LIN {X -0.007,Y -160.947,Z 1391.312,A 0.000,B 0.000,C 90.000,E1 236.135} C_DIS
LIN {X -0.022,Y -157.703,Z 1391.292,A 0.000,B 0.000,C 90.000,E1 232.603} C_DIS
LIN {X 0.041,Y -155.743,Z 1391.277,A 0.000,B 0.000,C 90.000,E1 229.908} C_DIS
LIN {X -0.013,Y -152.001,Z 1391.252,A 0.000,B 0.000,C 90.000,E1 225.445} C_DIS
LIN {X -0.001,Y -150.246,Z 1391.237,A 0.000,B 0.000,C 90.000,E1 222.732} C_DIS
LIN {X 0.031,Y -147.004,Z 1391.212,A 0.000,B 0.000,C 90.000,E1 218.177} C_DIS
LIN {X 0.021,Y -145.588,Z 1391.197,A 0.000,B 0.000,C 90.000,E1 215.438} C_DIS
LIN {X -0.058,Y -142.976,Z 1391.171,A 0.000,B 0.000,C 90.000,E1 210.875} C_DIS
LIN {X 0.069,Y -141.603,Z 1391.151,A 0.000,B 0.000,C 90.000,E1 207.129} C_DIS
LIN {X -0.017,Y -139.424,Z 1391.115,A 0.000,B 0.000,C 90.000,E1 200.663} C_DIS
LIN {X 0.035,Y -139.153,Z 1391.104,A 0.000,B 0.000,C 90.000,E1 198.779} C_DIS
LIN {X 0.057,Y -138.344,Z 1391.058,A 0.000,B 0.000,C 90.000,E1 190.366} C_DIS
LIN {X 0.043,Y -139.484,Z 1391.006,A 0.000,B 0.000,C 90.000,E1 181.031} C_DIS
LIN {X -0.017,Y -141.082,Z 1390.975,A 0.000,B 0.000,C 90.000,E1 175.469} C_DIS
LIN {X -0.063,Y -142.458,Z 1390.959,A 0.000,B 0.000,C 90.000,E1 172.704} C_DIS
LIN {X 0.027,Y -144.702,Z 1390.934,A 0.000,B 0.000,C 90.000,E1 168.049} C_DIS
LIN {X -0.021,Y -147.298,Z 1390.913,A 0.000,B 0.000,C 90.000,E1 164.393} C_DIS
LIN {X -0.007,Y -150.618,Z 1390.888,A 0.000,B 0.000,C 90.000,E1 159.826} C_DIS
LIN {X -0.071,Y -154.093,Z 1390.868,A 0.000,B 0.000,C 90.000,E1 156.230} C_DIS
LIN {X -0.006,Y -157.515,Z 1390.848,A 0.000,B 0.000,C 90.000,E1 152.615} C_DIS
LIN {X -0.061,Y -161.747,Z 1390.828,A 0.000,B 0.000,C 90.000,E1 149.076} C_DIS
LIN {X 0.045,Y -165.940,Z 1390.808,A 0.000,B 0.000,C 90.000,E1 145.515} C_DIS
LIN {X 0.043,Y -170.931,Z 1390.789,A 0.000,B 0.000,C 90.000,E1 142.029} C_DIS
LIN {X -0.037,Y -175.799,Z 1390.770,A 0.000,B 0.000,C 90.000,E1 138.609} C_DIS
LIN {X 0.091,Y -181.407,Z 1390.751,A 0.000,B 0.000,C 90.000,E1 135.162} C_DIS
LIN {X -0.034,Y -186.908,Z 1390.732,A 0.000,B 0.000,C 90.000,E1 131.838} C_DIS
LIN {X -0.082,Y -191.488,Z 1390.719,A 0.000,B 0.000,C 90.000,E1 129.358} C_DIS
LIN {X 0.125,Y -197.349,Z 1390.700,A 0.000,B 0.000,C 90.000,E1 126.011} C_DIS
LIN {X -0.018,Y -199.398,Z 1390.695,A 0.000,B 0.000,C 90.000,E1 125.025} C_DIS
LIN {X -0.063,Y -309.902,Z 1390.694,A 0.000,B 0.000,C 90.000,E1 125.025} C_DIS
LIN {X -0.002,Y -311.910,Z 1390.694,A 0.000,B 0.000,C 90.000,E1 124.978} C_DIS
LIN {X 0.038,Y -317.203,Z 1390.693,A 0.000,B 0.000,C 90.000,E1 124.692} C_DIS
LIN {X 0.080,Y -320.044,Z 1390.691,A 0.000,B 0.000,C 90.000,E1 124.405} C_DIS
LIN {X 0.017,Y -323.693,Z 1390.688,A 0.000,B 0.000,C 90.000,E1 123.865} C_DIS
LIN {X -0.171,Y -325.159,Z 1390.686,A 0.000,B 0.000,C 90.000,E1 123.579} C_DIS
LIN {X 0.060,Y -338.025,Z 1390.667,A 0.000,B 0.000,C 90.000,E1 120.079} C_DIS
LIN {X -0.098,Y -349.982,Z 1390.652,A 0.000,B 0.000,C 90.000,E1 117.334} C_DIS
LIN {X 0.073,Y -363.402,Z 1390.637,A 0.000,B 0.000,C 90.000,E1 114.591} C_DIS
LIN {X 0.224,Y -376.645,Z 1390.624,A 0.000,B 0.000,C 90.000,E1 112.206} C_DIS
LIN {X -0.078,Y -391.224,Z 1390.611,A 0.000,B 0.000,C 90.000,E1 109.939} C_DIS
LIN {X -0.169,Y -407.239,Z 1390.598,A 0.000,B 0.000,C 90.000,E1 107.692} C_DIS
LIN {X -0.119,Y -424.803,Z 1390.586,A 0.000,B 0.000,C 90.000,E1 105.481} C_DIS
LIN {X 0.188,Y -444.001,Z 1390.574,A 0.000,B 0.000,C 90.000,E1 103.300} C_DIS
LIN {X 0.222,Y -464.106,Z 1390.563,A 0.000,B 0.000,C 90.000,E1 101.299} C_DIS
LIN {X -0.112,Y -482.128,Z 1390.554,A 0.000,B 0.000,C 90.000,E1 99.726} C_DIS
LIN {X -0.082,Y -484.477,Z 1390.553,A 0.000,B 0.000,C 90.000,E1 99.500} C_DIS
LIN {X -0.092,Y -486.349,Z 1390.551,A 0.000,B 0.000,C 90.000,E1 99.265} C_DIS
LIN {X -0.103,Y -487.770,Z 1390.550,A 0.000,B 0.000,C 90.000,E1 99.029} C_DIS
LIN {X 0.094,Y -489.689,Z 1390.547,A 0.000,B 0.000,C 90.000,E1 98.511} C_DIS
LIN {X -0.183,Y -490.477,Z 1390.545,A 0.000,B 0.000,C 90.000,E1 98.049} C_DIS
LIN {X 0.039,Y -490.272,Z 1390.542,A 0.000,B 0.000,C 90.000,E1 97.530} C_DIS
LIN {X -0.220,Y -489.046,Z 1390.539,A 0.000,B 0.000,C 90.000,E1 97.068} C_DIS
LIN {X 0.164,Y -487.991,Z 1390.538,A 0.000,B 0.000,C 90.000,E1 96.777} C_DIS
LIN {X 0.006,Y -486.568,Z 1390.536,A 0.000,B 0.000,C 90.000,E1 96.549} C_DIS
LIN {X 0.174,Y -468.415,Z 1390.521,A 0.000,B 0.000,C 90.000,E1 93.784} C_DIS
LIN {X 0.105,Y -460.162,Z 1390.514,A 0.000,B 0.000,C 90.000,E1 92.522} C_DIS
LIN {X 0.170,Y -439.101,Z 1390.495,A 0.000,B 0.000,C 90.000,E1 89.141} C_DIS
LIN {X 0.130,Y -427.055,Z 1390.484,A 0.000,B 0.000,C 90.000,E1 87.020} C_DIS
LIN {X 0.051,Y -417.995,Z 1390.475,A 0.000,B 0.000,C 90.000,E1 85.412} C_DIS
LIN {X -0.076,Y -407.198,Z 1390.464,A 0.000,B 0.000,C 90.000,E1 83.514} C_DIS
LIN {X -0.007,Y -397.916,Z 1390.455,A 0.000,B 0.000,C 90.000,E1 81.837} C_DIS
LIN {X -0.041,Y -388.423,Z 1390.445,A 0.000,B 0.000,C 90.000,E1 80.151} C_DIS
LIN {X 0.150,Y -377.105,Z 1390.434,A 0.000,B 0.000,C 90.000,E1 78.117} C_DIS
LIN {X -0.100,Y -367.376,Z 1390.424,A 0.000,B 0.000,C 90.000,E1 76.408} C_DIS
LIN {X -0.068,Y -357.511,Z 1390.415,A 0.000,B 0.000,C 90.000,E1 74.629} C_DIS
LIN {X 0.139,Y -345.870,Z 1390.403,A 0.000,B 0.000,C 90.000,E1 72.489} C_DIS
LIN {X -0.034,Y -334.159,Z 1390.391,A 0.000,B 0.000,C 90.000,E1 70.369} C_DIS
LIN {X 0.000,Y -319.385,Z 1390.375,A 0.000,B 0.000,C 90.000,E1 67.539} C_DIS
LIN {X -0.087,Y -304.192,Z 1390.357,A 0.000,B 0.000,C 90.000,E1 64.332} C_DIS
LIN {X -0.089,Y -294.606,Z 1390.344,A 0.000,B 0.000,C 90.000,E1 62.025} C_DIS
LIN {X -0.064,Y -283.523,Z 1390.328,A 0.000,B 0.000,C 90.000,E1 58.997} C_DIS
LIN {X 0.029,Y -272.556,Z 1390.309,A 0.000,B 0.000,C 90.000,E1 55.548} C_DIS
LIN {X 0.000,Y -264.344,Z 1390.293,A 0.000,B 0.000,C 90.000,E1 52.763} C_DIS
LIN {X -0.022,Y -254.665,Z 1390.273,A 0.000,B 0.000,C 90.000,E1 49.218} C_DIS
LIN {X 0.126,Y -245.587,Z 1390.253,A 0.000,B 0.000,C 90.000,E1 45.567} C_DIS
LIN {X -0.016,Y -237.338,Z 1390.233,A 0.000,B 0.000,C 90.000,E1 41.919} C_DIS
LIN {X -0.014,Y -229.913,Z 1390.212,A 0.000,B 0.000,C 90.000,E1 38.177} C_DIS
LIN {X -0.119,Y -223.465,Z 1390.191,A 0.000,B 0.000,C 90.000,E1 34.405} C_DIS
LIN {X -0.057,Y -217.896,Z 1390.170,A 0.000,B 0.000,C 90.000,E1 30.541} C_DIS
LIN {X 0.065,Y -213.211,Z 1390.148,A 0.000,B 0.000,C 90.000,E1 26.616} C_DIS
LIN {X 0.062,Y -208.925,Z 1390.122,A 0.000,B 0.000,C 90.000,E1 21.897} C_DIS
LIN {X -0.044,Y -205.454,Z 1390.091,A 0.000,B 0.000,C 90.000,E1 16.370} C_DIS
LIN {X 0.036,Y -203.518,Z 1390.069,A 0.000,B 0.000,C 90.000,E1 12.355} C_DIS
LIN {X 0.051,Y -201.769,Z 1390.046,A 0.000,B 0.000,C 90.000,E1 8.341} C_DIS
LIN {X 0.093,Y -200.092,Z 1390.020,A 0.000,B 0.000,C 90.000,E1 3.498} C_DIS
LIN {X -0.036,Y -199.010,Z 1389.997,A 0.000,B 0.000,C 90.000,E1 359.542} C_DIS
LIN {X 0.026,Y -198.200,Z 1389.970,A 0.000,B 0.000,C 90.000,E1 354.666} C_DIS
LIN {X 0.019,Y -198.275,Z 1389.943,A 0.000,B 0.000,C 90.000,E1 349.803} C_DIS
LIN {X -0.076,Y -200.441,Z 1389.903,A 0.000,B 0.000,C 90.000,E1 342.543} C_DIS
LIN {X 0.078,Y -203.482,Z 1389.876,A 0.000,B 0.000,C 90.000,E1 337.667} C_DIS
LIN {X -0.013,Y -207.221,Z 1389.854,A 0.000,B 0.000,C 90.000,E1 333.691} C_DIS
LIN {X -0.081,Y -212.111,Z 1389.832,A 0.000,B 0.000,C 90.000,E1 329.744} C_DIS
LIN {X -0.001,Y -216.931,Z 1389.814,A 0.000,B 0.000,C 90.000,E1 326.580} C_DIS
LIN {X -0.103,Y -222.588,Z 1389.797,A 0.000,B 0.000,C 90.000,E1 323.497} C_DIS
LIN {X -0.006,Y -229.169,Z 1389.780,A 0.000,B 0.000,C 90.000,E1 320.400} C_DIS
LIN {X 0.033,Y -237.647,Z 1389.761,A 0.000,B 0.000,C 90.000,E1 316.986} C_DIS
LIN {X 0.139,Y -247.089,Z 1389.743,A 0.000,B 0.000,C 90.000,E1 313.623} C_DIS
LIN {X -0.010,Y -256.632,Z 1389.726,A 0.000,B 0.000,C 90.000,E1 310.744} C_DIS
LIN {X -0.025,Y -267.405,Z 1389.710,A 0.000,B 0.000,C 90.000,E1 307.890} C_DIS
LIN {X -0.082,Y -279.297,Z 1389.695,A 0.000,B 0.000,C 90.000,E1 305.105} C_DIS
LIN {X 0.002,Y -287.678,Z 1389.685,A 0.000,B 0.000,C 90.000,E1 303.372} C_DIS
LIN {X 0.070,Y -295.164,Z 1389.678,A 0.000,B 0.000,C 90.000,E1 302.005} C_DIS
LIN {X 0.080,Y -303.455,Z 1389.670,A 0.000,B 0.000,C 90.000,E1 300.669} C_DIS
LIN {X 0.043,Y -312.546,Z 1389.663,A 0.000,B 0.000,C 90.000,E1 299.361} C_DIS
LIN {X -0.065,Y -325.434,Z 1389.654,A 0.000,B 0.000,C 90.000,E1 297.769} C_DIS
LIN {X -0.150,Y -344.025,Z 1389.643,A 0.000,B 0.000,C 90.000,E1 295.720} C_DIS
LIN {X -0.082,Y -357.370,Z 1389.635,A 0.000,B 0.000,C 90.000,E1 294.259} C_DIS
LIN {X -0.075,Y -370.622,Z 1389.627,A 0.000,B 0.000,C 90.000,E1 292.823} C_DIS
LIN {X 0.032,Y -380.903,Z 1389.620,A 0.000,B 0.000,C 90.000,E1 291.663} C_DIS
LIN {X -0.089,Y -393.414,Z 1389.612,A 0.000,B 0.000,C 90.000,E1 290.248} C_DIS
LIN {X -0.210,Y -415.670,Z 1389.599,A 0.000,B 0.000,C 90.000,E1 287.764} C_DIS
LIN {X -0.005,Y -423.043,Z 1389.594,A 0.000,B 0.000,C 90.000,E1 286.913} C_DIS
LIN {X 0.151,Y -429.812,Z 1389.589,A 0.000,B 0.000,C 90.000,E1 286.079} C_DIS
LIN {X -0.052,Y -435.857,Z 1389.585,A 0.000,B 0.000,C 90.000,E1 285.300} C_DIS
LIN {X 0.112,Y -441.130,Z 1389.581,A 0.000,B 0.000,C 90.000,E1 284.481} C_DIS
LIN {X 0.002,Y -445.562,Z 1389.576,A 0.000,B 0.000,C 90.000,E1 283.703} C_DIS
LIN {X -0.174,Y -449.126,Z 1389.572,A 0.000,B 0.000,C 90.000,E1 282.939} C_DIS
LIN {X 0.065,Y -450.175,Z 1389.570,A 0.000,B 0.000,C 90.000,E1 282.647} C_DIS
LIN {X 0.118,Y -451.960,Z 1389.567,A 0.000,B 0.000,C 90.000,E1 282.119} C_DIS
LIN {X 0.176,Y -453.382,Z 1389.565,A 0.000,B 0.000,C 90.000,E1 281.591} C_DIS
LIN {X 0.158,Y -454.432,Z 1389.562,A 0.000,B 0.000,C 90.000,E1 281.074} C_DIS
LIN {X -0.211,Y -455.103,Z 1389.559,A 0.000,B 0.000,C 90.000,E1 280.602} C_DIS
LIN {X -0.129,Y -455.379,Z 1389.556,A 0.000,B 0.000,C 90.000,E1 280.074} C_DIS
LIN {X -0.122,Y -455.153,Z 1389.553,A 0.000,B 0.000,C 90.000,E1 279.557} C_DIS
LIN {X -0.039,Y -454.522,Z 1389.550,A 0.000,B 0.000,C 90.000,E1 279.029} C_DIS
LIN {X -0.029,Y -453.394,Z 1389.547,A 0.000,B 0.000,C 90.000,E1 278.511} C_DIS
LIN {X -0.019,Y -451.742,Z 1389.544,A 0.000,B 0.000,C 90.000,E1 277.992} C_DIS
LIN {X 0.045,Y -449.474,Z 1389.542,A 0.000,B 0.000,C 90.000,E1 277.466} C_DIS
LIN {X 0.032,Y -446.487,Z 1389.539,A 0.000,B 0.000,C 90.000,E1 276.947} C_DIS
LIN {X -0.229,Y -444.735,Z 1389.537,A 0.000,B 0.000,C 90.000,E1 276.720} C_DIS
LIN {X 0.176,Y -440.474,Z 1389.534,A 0.000,B 0.000,C 90.000,E1 276.144} C_DIS
LIN {X 0.162,Y -435.121,Z 1389.531,A 0.000,B 0.000,C 90.000,E1 275.625} C_DIS
LIN {X -0.011,Y -429.033,Z 1389.529,A 0.000,B 0.000,C 90.000,E1 275.163} C_DIS
LIN {X -0.162,Y -422.710,Z 1389.526,A 0.000,B 0.000,C 90.000,E1 274.759} C_DIS
LIN {X 0.039,Y -416.084,Z 1389.524,A 0.000,B 0.000,C 90.000,E1 274.359} C_DIS
LIN {X 0.186,Y -409.418,Z 1389.522,A 0.000,B 0.000,C 90.000,E1 274.012} C_DIS
LIN {X 0.002,Y -399.432,Z 1389.520,A 0.000,B 0.000,C 90.000,E1 273.612} C_DIS
LIN {X -0.163,Y -392.867,Z 1389.519,A 0.000,B 0.000,C 90.000,E1 273.383} C_DIS
LIN {X -0.075,Y -379.503,Z 1389.516,A 0.000,B 0.000,C 90.000,E1 272.922} C_DIS
LIN {X 0.119,Y -372.448,Z 1389.515,A 0.000,B 0.000,C 90.000,E1 272.694} C_DIS
LIN {X 0.115,Y -364.946,Z 1389.514,A 0.000,B 0.000,C 90.000,E1 272.522} C_DIS
LIN {X -0.074,Y -353.742,Z 1389.513,A 0.000,B 0.000,C 90.000,E1 272.350} C_DIS
LIN {X -0.043,Y -344.232,Z 1389.512,A 0.000,B 0.000,C 90.000,E1 272.236} C_DIS
LIN {X -0.006,Y -329.258,Z 1389.512,A 0.000,B 0.000,C 90.000,E1 272.121} C_DIS
LIN {X -0.119,Y -323.444,Z 1389.512,A 0.000,B 0.000,C 90.000,E1 272.121} C_DIS
LIN {X -0.091,Y -181.247,Z 1389.512,A 0.000,B 0.000,C 90.000,E1 272.121} C_DIS
LIN {X 0.034,Y -181.578,Z 1389.502,A 0.000,B 0.000,C 90.000,E1 270.344} C_DIS
LIN {X 0.009,Y -180.904,Z 1389.474,A 0.000,B 0.000,C 90.000,E1 265.298} C_DIS
LIN {X -0.041,Y -180.245,Z 1389.464,A 0.000,B 0.000,C 90.000,E1 263.628} C_DIS
LIN {X -0.022,Y -178.732,Z 1389.441,A 0.000,B 0.000,C 90.000,E1 259.398} C_DIS
LIN {X 0.046,Y -175.780,Z 1389.413,A 0.000,B 0.000,C 90.000,E1 254.283} C_DIS
LIN {X 0.033,Y -171.964,Z 1389.384,A 0.000,B 0.000,C 90.000,E1 249.156} C_DIS
LIN {X 0.070,Y -171.361,Z 1389.380,A 0.000,B 0.000,C 90.000,E1 248.284} C_DIS
LIN {X 0.048,Y -167.610,Z 1389.355,A 0.000,B 0.000,C 90.000,E1 243.973} C_DIS
LIN {X 0.060,Y -166.257,Z 1389.346,A 0.000,B 0.000,C 90.000,E1 242.231} C_DIS
LIN {X 0.047,Y -163.011,Z 1389.326,A 0.000,B 0.000,C 90.000,E1 238.742} C_DIS
LIN {X -0.040,Y -160.934,Z 1389.312,A 0.000,B 0.000,C 90.000,E1 236.135} C_DIS
LIN {X 0.071,Y -157.694,Z 1389.292,A 0.000,B 0.000,C 90.000,E1 232.557} C_DIS
LIN {X 0.008,Y -155.734,Z 1389.277,A 0.000,B 0.000,C 90.000,E1 229.908} C_DIS
LIN {X 0.061,Y -151.992,Z 1389.252,A 0.000,B 0.000,C 90.000,E1 225.405} C_DIS
LIN {X 0.078,Y -150.236,Z 1389.237,A 0.000,B 0.000,C 90.000,E1 222.690} C_DIS
LIN {X 0.001,Y -146.996,Z 1389.212,A 0.000,B 0.000,C 90.000,E1 218.177} C_DIS
LIN {X -0.009,Y -145.581,Z 1389.197,A 0.000,B 0.000,C 90.000,E1 215.438} C_DIS
LIN {X -0.015,Y -142.970,Z 1389.171,A 0.000,B 0.000,C 90.000,E1 210.846} C_DIS
LIN {X 0.038,Y -141.597,Z 1389.151,A 0.000,B 0.000,C 90.000,E1 207.129} C_DIS
LIN {X -0.046,Y -139.422,Z 1389.115,A 0.000,B 0.000,C 90.000,E1 200.663} C_DIS
LIN {X 0.005,Y -139.149,Z 1389.104,A 0.000,B 0.000,C 90.000,E1 198.779} C_DIS
LIN {X 0.027,Y -138.345,Z 1389.058,A 0.000,B 0.000,C 90.000,E1 190.366} C_DIS
LIN {X 0.013,Y -139.487,Z 1389.006,A 0.000,B 0.000,C 90.000,E1 181.031} C_DIS
LIN {X -0.048,Y -141.088,Z 1388.975,A 0.000,B 0.000,C 90.000,E1 175.469} C_DIS
LIN {X 0.048,Y -142.464,Z 1388.959,A 0.000,B 0.000,C 90.000,E1 172.648} C_DIS
LIN {X -0.004,Y -144.709,Z 1388.934,A 0.000,B 0.000,C 90.000,E1 168.049} C_DIS
LIN {X -0.053,Y -147.307,Z 1388.913,A 0.000,B 0.000,C 90.000,E1 164.393} C_DIS
LIN {X -0.038,Y -150.628,Z 1388.888,A 0.000,B 0.000,C 90.000,E1 159.826} C_DIS
LIN {X 0.038,Y -154.105,Z 1388.868,A 0.000,B 0.000,C 90.000,E1 156.177} C_DIS
LIN {X -0.038,Y -157.528,Z 1388.848,A 0.000,B 0.000,C 90.000,E1 152.615} C_DIS
LIN {X -0.094,Y -161.763,Z 1388.828,A 0.000,B 0.000,C 90.000,E1 149.076} C_DIS
LIN {X 0.012,Y -165.956,Z 1388.808,A 0.000,B 0.000,C 90.000,E1 145.515} C_DIS
LIN {X 0.008,Y -170.948,Z 1388.789,A 0.000,B 0.000,C 90.000,E1 142.029} C_DIS
LIN {X -0.072,Y -175.816,Z 1388.770,A 0.000,B 0.000,C 90.000,E1 138.609} C_DIS
LIN {X 0.056,Y -181.424,Z 1388.751,A 0.000,B 0.000,C 90.000,E1 135.162} C_DIS
LIN {X -0.070,Y -186.928,Z 1388.732,A 0.000,B 0.000,C 90.000,E1 131.838} C_DIS
LIN {X 0.003,Y -191.505,Z 1388.719,A 0.000,B 0.000,C 90.000,E1 129.322} C_DIS
LIN {X 0.087,Y -197.370,Z 1388.700,A 0.000,B 0.000,C 90.000,E1 126.011} C_DIS
LIN {X 0.013,Y -199.380,Z 1388.695,A 0.000,B 0.000,C 90.000,E1 125.025} C_DIS
LIN {X -0.015,Y -310.039,Z 1388.695,A 0.000,B 0.000,C 90.000,E1 125.025} C_DIS
LIN {X -0.060,Y -312.563,Z 1388.694,A 0.000,B 0.000,C 90.000,E1 124.978} C_DIS
LIN {X -0.021,Y -317.410,Z 1388.693,A 0.000,B 0.000,C 90.000,E1 124.692} C_DIS
LIN {X 0.020,Y -320.169,Z 1388.691,A 0.000,B 0.000,C 90.000,E1 124.405} C_DIS
LIN {X 0.044,Y -322.213,Z 1388.690,A 0.000,B 0.000,C 90.000,E1 124.119} C_DIS
LIN {X 0.066,Y -323.810,Z 1388.688,A 0.000,B 0.000,C 90.000,E1 123.833} C_DIS
LIN {X 0.155,Y -325.234,Z 1388.686,A 0.000,B 0.000,C 90.000,E1 123.499} C_DIS
LIN {X -0.062,Y -338.085,Z 1388.667,A 0.000,B 0.000,C 90.000,E1 120.079} C_DIS
LIN {X -0.061,Y -350.054,Z 1388.652,A 0.000,B 0.000,C 90.000,E1 117.308} C_DIS
LIN {X -0.052,Y -363.484,Z 1388.637,A 0.000,B 0.000,C 90.000,E1 114.591} C_DIS
LIN {X 0.096,Y -376.738,Z 1388.623,A 0.000,B 0.000,C 90.000,E1 112.206} C_DIS
LIN {X -0.209,Y -391.327,Z 1388.611,A 0.000,B 0.000,C 90.000,E1 109.939} C_DIS
LIN {X 0.086,Y -407.354,Z 1388.598,A 0.000,B 0.000,C 90.000,E1 107.638} C_DIS
LIN {X 0.154,Y -424.932,Z 1388.586,A 0.000,B 0.000,C 90.000,E1 105.426} C_DIS
LIN {X 0.050,Y -444.142,Z 1388.574,A 0.000,B 0.000,C 90.000,E1 103.300} C_DIS
LIN {X 0.089,Y -464.252,Z 1388.563,A 0.000,B 0.000,C 90.000,E1 101.299} C_DIS
LIN {X 0.234,Y -482.276,Z 1388.554,A 0.000,B 0.000,C 90.000,E1 99.670} C_DIS
LIN {X -0.211,Y -484.555,Z 1388.553,A 0.000,B 0.000,C 90.000,E1 99.500} C_DIS
LIN {X 0.223,Y -486.400,Z 1388.551,A 0.000,B 0.000,C 90.000,E1 99.208} C_DIS
LIN {X 0.176,Y -487.796,Z 1388.550,A 0.000,B 0.000,C 90.000,E1 98.973} C_DIS
LIN {X -0.108,Y -489.627,Z 1388.547,A 0.000,B 0.000,C 90.000,E1 98.511} C_DIS
LIN {X 0.100,Y -490.347,Z 1388.544,A 0.000,B 0.000,C 90.000,E1 97.992} C_DIS
LIN {X -0.165,Y -490.076,Z 1388.542,A 0.000,B 0.000,C 90.000,E1 97.530} C_DIS
LIN {X 0.122,Y -488.776,Z 1388.539,A 0.000,B 0.000,C 90.000,E1 97.004} C_DIS
LIN {X -0.039,Y -487.675,Z 1388.538,A 0.000,B 0.000,C 90.000,E1 96.777} C_DIS
LIN {X 0.176,Y -484.470,Z 1388.535,A 0.000,B 0.000,C 90.000,E1 96.258} C_DIS
LIN {X -0.033,Y -468.028,Z 1388.521,A 0.000,B 0.000,C 90.000,E1 93.784} C_DIS
LIN {X 0.137,Y -458.042,Z 1388.513,A 0.000,B 0.000,C 90.000,E1 92.236} C_DIS
LIN {X -0.045,Y -438.754,Z 1388.495,A 0.000,B 0.000,C 90.000,E1 89.141} C_DIS
LIN {X -0.087,Y -426.719,Z 1388.483,A 0.000,B 0.000,C 90.000,E1 87.020} C_DIS
LIN {X -0.166,Y -417.674,Z 1388.474,A 0.000,B 0.000,C 90.000,E1 85.412} C_DIS
LIN {X 0.110,Y -406.907,Z 1388.464,A 0.000,B 0.000,C 90.000,E1 83.457} C_DIS
LIN {X 0.168,Y -397.627,Z 1388.454,A 0.000,B 0.000,C 90.000,E1 81.781} C_DIS
LIN {X 0.124,Y -388.165,Z 1388.445,A 0.000,B 0.000,C 90.000,E1 80.095} C_DIS
LIN {X -0.067,Y -376.860,Z 1388.434,A 0.000,B 0.000,C 90.000,E1 78.117} C_DIS
LIN {X 0.041,Y -367.109,Z 1388.424,A 0.000,B 0.000,C 90.000,E1 76.353} C_DIS
LIN {X 0.061,Y -357.247,Z 1388.414,A 0.000,B 0.000,C 90.000,E1 74.574} C_DIS
LIN {X -0.075,Y -345.598,Z 1388.403,A 0.000,B 0.000,C 90.000,E1 72.489} C_DIS
LIN {X 0.191,Y -335.551,Z 1388.392,A 0.000,B 0.000,C 90.000,E1 70.604} C_DIS
LIN {X 0.134,Y -320.732,Z 1388.377,A 0.000,B 0.000,C 90.000,E1 67.794} C_DIS
LIN {X 0.076,Y -305.397,Z 1388.359,A 0.000,B 0.000,C 90.000,E1 64.588} C_DIS
LIN {X 0.098,Y -295.693,Z 1388.346,A 0.000,B 0.000,C 90.000,E1 62.281} C_DIS
LIN {X -0.002,Y -284.507,Z 1388.329,A 0.000,B 0.000,C 90.000,E1 59.282} C_DIS
LIN {X -0.052,Y -274.549,Z 1388.312,A 0.000,B 0.000,C 90.000,E1 56.215} C_DIS
LIN {X 0.034,Y -266.283,Z 1388.297,A 0.000,B 0.000,C 90.000,E1 53.417} C_DIS
LIN {X -0.095,Y -256.516,Z 1388.277,A 0.000,B 0.000,C 90.000,E1 49.908} C_DIS
LIN {X 0.101,Y -249.122,Z 1388.261,A 0.000,B 0.000,C 90.000,E1 46.986} C_DIS
LIN {X 0.065,Y -240.559,Z 1388.241,A 0.000,B 0.000,C 90.000,E1 43.338} C_DIS
LIN {X -0.037,Y -232.821,Z 1388.220,A 0.000,B 0.000,C 90.000,E1 39.644} C_DIS
LIN {X -0.100,Y -225.988,Z 1388.199,A 0.000,B 0.000,C 90.000,E1 35.884} C_DIS
LIN {X 0.095,Y -220.105,Z 1388.178,A 0.000,B 0.000,C 90.000,E1 32.005} C_DIS
LIN {X 0.008,Y -215.100,Z 1388.156,A 0.000,B 0.000,C 90.000,E1 28.153} C_DIS
LIN {X -0.030,Y -210.411,Z 1388.130,A 0.000,B 0.000,C 90.000,E1 23.462} C_DIS
LIN {X -0.051,Y -206.577,Z 1388.099,A 0.000,B 0.000,C 90.000,E1 17.928} C_DIS
LIN {X -0.031,Y -204.541,Z 1388.077,A 0.000,B 0.000,C 90.000,E1 13.939} C_DIS
LIN {X 0.086,Y -202.702,Z 1388.055,A 0.000,B 0.000,C 90.000,E1 9.905} C_DIS
LIN {X 0.010,Y -201.112,Z 1388.033,A 0.000,B 0.000,C 90.000,E1 5.910} C_DIS
LIN {X -0.032,Y -199.864,Z 1388.010,A 0.000,B 0.000,C 90.000,E1 1.892} C_DIS
LIN {X 0.094,Y -198.715,Z 1387.984,A 0.000,B 0.000,C 90.000,E1 357.078} C_DIS
LIN {X 0.004,Y -198.368,Z 1387.952,A 0.000,B 0.000,C 90.000,E1 351.432} C_DIS
LIN {X 0.050,Y -200.274,Z 1387.907,A 0.000,B 0.000,C 90.000,E1 343.323} C_DIS
LIN {X -0.076,Y -203.693,Z 1387.876,A 0.000,B 0.000,C 90.000,E1 337.720} C_DIS
LIN {X 0.030,Y -207.426,Z 1387.854,A 0.000,B 0.000,C 90.000,E1 333.691} C_DIS
LIN {X -0.031,Y -212.322,Z 1387.832,A 0.000,B 0.000,C 90.000,E1 329.744} C_DIS
LIN {X 0.054,Y -217.141,Z 1387.814,A 0.000,B 0.000,C 90.000,E1 326.580} C_DIS
LIN {X -0.040,Y -222.807,Z 1387.797,A 0.000,B 0.000,C 90.000,E1 323.497} C_DIS
LIN {X -0.082,Y -229.358,Z 1387.780,A 0.000,B 0.000,C 90.000,E1 320.436} C_DIS
LIN {X -0.050,Y -237.819,Z 1387.761,A 0.000,B 0.000,C 90.000,E1 317.025} C_DIS
LIN {X -0.123,Y -247.240,Z 1387.743,A 0.000,B 0.000,C 90.000,E1 313.704} C_DIS
LIN {X -0.085,Y -256.762,Z 1387.726,A 0.000,B 0.000,C 90.000,E1 310.782} C_DIS
LIN {X 0.076,Y -267.503,Z 1387.711,A 0.000,B 0.000,C 90.000,E1 307.890} C_DIS
LIN {X 0.025,Y -279.395,Z 1387.695,A 0.000,B 0.000,C 90.000,E1 305.105} C_DIS
LIN {X 0.148,Y -285.995,Z 1387.687,A 0.000,B 0.000,C 90.000,E1 303.706} C_DIS
LIN {X -0.063,Y -295.238,Z 1387.678,A 0.000,B 0.000,C 90.000,E1 302.054} C_DIS
LIN {X -0.060,Y -303.486,Z 1387.671,A 0.000,B 0.000,C 90.000,E1 300.718} C_DIS
LIN {X -0.105,Y -312.592,Z 1387.663,A 0.000,B 0.000,C 90.000,E1 299.411} C_DIS
LIN {X 0.074,Y -325.439,Z 1387.654,A 0.000,B 0.000,C 90.000,E1 297.769} C_DIS
LIN {X -0.034,Y -344.012,Z 1387.643,A 0.000,B 0.000,C 90.000,E1 295.720} C_DIS
LIN {X 0.079,Y -357.274,Z 1387.635,A 0.000,B 0.000,C 90.000,E1 294.259} C_DIS
LIN {X 0.100,Y -370.493,Z 1387.627,A 0.000,B 0.000,C 90.000,E1 292.823} C_DIS
LIN {X -0.138,Y -380.766,Z 1387.620,A 0.000,B 0.000,C 90.000,E1 291.716} C_DIS
LIN {X -0.082,Y -390.849,Z 1387.614,A 0.000,B 0.000,C 90.000,E1 290.556} C_DIS
LIN {X 0.166,Y -413.151,Z 1387.600,A 0.000,B 0.000,C 90.000,E1 288.000} C_DIS
LIN {X 0.094,Y -423.000,Z 1387.594,A 0.000,B 0.000,C 90.000,E1 286.913} C_DIS
LIN {X -0.161,Y -429.795,Z 1387.589,A 0.000,B 0.000,C 90.000,E1 286.134} C_DIS
LIN {X 0.048,Y -435.854,Z 1387.585,A 0.000,B 0.000,C 90.000,E1 285.300} C_DIS
LIN {X -0.213,Y -441.167,Z 1387.581,A 0.000,B 0.000,C 90.000,E1 284.537} C_DIS
LIN {X -0.219,Y -444.260,Z 1387.578,A 0.000,B 0.000,C 90.000,E1 284.008} C_DIS
LIN {X 0.129,Y -448.162,Z 1387.573,A 0.000,B 0.000,C 90.000,E1 283.175} C_DIS
LIN {X 0.170,Y -450.333,Z 1387.570,A 0.000,B 0.000,C 90.000,E1 282.647} C_DIS
LIN {X 0.224,Y -452.123,Z 1387.568,A 0.000,B 0.000,C 90.000,E1 282.119} C_DIS
LIN {X -0.251,Y -453.580,Z 1387.565,A 0.000,B 0.000,C 90.000,E1 281.658} C_DIS
LIN {X -0.180,Y -454.638,Z 1387.562,A 0.000,B 0.000,C 90.000,E1 281.130} C_DIS
LIN {X -0.101,Y -455.320,Z 1387.559,A 0.000,B 0.000,C 90.000,E1 280.602} C_DIS
LIN {X -0.018,Y -455.611,Z 1387.556,A 0.000,B 0.000,C 90.000,E1 280.074} C_DIS
LIN {X -0.010,Y -455.430,Z 1387.553,A 0.000,B 0.000,C 90.000,E1 279.557} C_DIS
LIN {X 0.074,Y -454.801,Z 1387.550,A 0.000,B 0.000,C 90.000,E1 279.029} C_DIS
LIN {X 0.086,Y -453.719,Z 1387.547,A 0.000,B 0.000,C 90.000,E1 278.511} C_DIS
LIN {X 0.097,Y -452.061,Z 1387.544,A 0.000,B 0.000,C 90.000,E1 277.992} C_DIS
LIN {X 0.104,Y -449.841,Z 1387.542,A 0.000,B 0.000,C 90.000,E1 277.473} C_DIS
LIN {X 0.150,Y -446.930,Z 1387.539,A 0.000,B 0.000,C 90.000,E1 276.947} C_DIS
LIN {X -0.109,Y -445.238,Z 1387.537,A 0.000,B 0.000,C 90.000,E1 276.720} C_DIS
LIN {X -0.140,Y -441.050,Z 1387.534,A 0.000,B 0.000,C 90.000,E1 276.201} C_DIS
LIN {X -0.182,Y -435.811,Z 1387.531,A 0.000,B 0.000,C 90.000,E1 275.682} C_DIS
LIN {X 0.033,Y -432.760,Z 1387.530,A 0.000,B 0.000,C 90.000,E1 275.391} C_DIS
LIN {X 0.000,Y -426.500,Z 1387.527,A 0.000,B 0.000,C 90.000,E1 274.935} C_DIS
LIN {X -0.001,Y -420.045,Z 1387.525,A 0.000,B 0.000,C 90.000,E1 274.531} C_DIS
LIN {X -0.034,Y -413.423,Z 1387.523,A 0.000,B 0.000,C 90.000,E1 274.188} C_DIS
LIN {X 0.095,Y -403.586,Z 1387.521,A 0.000,B 0.000,C 90.000,E1 273.726} C_DIS
LIN {X 0.170,Y -393.766,Z 1387.519,A 0.000,B 0.000,C 90.000,E1 273.326} C_DIS
LIN {X 0.187,Y -383.714,Z 1387.517,A 0.000,B 0.000,C 90.000,E1 272.980} C_DIS
LIN {X 0.056,Y -373.320,Z 1387.515,A 0.000,B 0.000,C 90.000,E1 272.694} C_DIS
LIN {X 0.061,Y -365.993,Z 1387.514,A 0.000,B 0.000,C 90.000,E1 272.522} C_DIS
LIN {X -0.142,Y -354.681,Z 1387.513,A 0.000,B 0.000,C 90.000,E1 272.350} C_DIS
LIN {X -0.114,Y -345.263,Z 1387.512,A 0.000,B 0.000,C 90.000,E1 272.236} C_DIS
LIN {X -0.067,Y -330.692,Z 1387.512,A 0.000,B 0.000,C 90.000,E1 272.121} C_DIS
LIN {X 0.104,Y -321.131,Z 1387.512,A 0.000,B 0.000,C 90.000,E1 272.064} C_DIS
LIN {X 0.035,Y -181.250,Z 1387.511,A 0.000,B 0.000,C 90.000,E1 272.064} C_DIS
LIN {X 0.003,Y -181.579,Z 1387.502,A 0.000,B 0.000,C 90.000,E1 270.344} C_DIS
LIN {X -0.021,Y -180.904,Z 1387.474,A 0.000,B 0.000,C 90.000,E1 265.298} C_DIS
LIN {X -0.071,Y -180.240,Z 1387.464,A 0.000,B 0.000,C 90.000,E1 263.628} C_DIS
LIN {X -0.052,Y -178.727,Z 1387.441,A 0.000,B 0.000,C 90.000,E1 259.398} C_DIS
LIN {X 0.015,Y -175.775,Z 1387.413,A 0.000,B 0.000,C 90.000,E1 254.283} C_DIS
LIN {X 0.003,Y -171.958,Z 1387.384,A 0.000,B 0.000,C 90.000,E1 249.156} C_DIS
LIN {X 0.041,Y -171.352,Z 1387.379,A 0.000,B 0.000,C 90.000,E1 248.284} C_DIS
LIN {X 0.019,Y -167.603,Z 1387.355,A 0.000,B 0.000,C 90.000,E1 243.973} C_DIS
LIN {X 0.031,Y -166.247,Z 1387.346,A 0.000,B 0.000,C 90.000,E1 242.231} C_DIS
LIN {X 0.019,Y -163.003,Z 1387.326,A 0.000,B 0.000,C 90.000,E1 238.742} C_DIS
LIN {X 0.065,Y -160.924,Z 1387.312,A 0.000,B 0.000,C 90.000,E1 236.087} C_DIS
LIN {X 0.043,Y -157.685,Z 1387.292,A 0.000,B 0.000,C 90.000,E1 232.557} C_DIS
LIN {X -0.019,Y -155.726,Z 1387.277,A 0.000,B 0.000,C 90.000,E1 229.908} C_DIS
LIN {X 0.035,Y -151.985,Z 1387.252,A 0.000,B 0.000,C 90.000,E1 225.405} C_DIS
LIN {X 0.051,Y -150.229,Z 1387.237,A 0.000,B 0.000,C 90.000,E1 222.690} C_DIS
LIN {X -0.026,Y -146.990,Z 1387.212,A 0.000,B 0.000,C 90.000,E1 218.177} C_DIS
LIN {X -0.035,Y -145.576,Z 1387.197,A 0.000,B 0.000,C 90.000,E1 215.438} C_DIS
LIN {X 0.081,Y -142.965,Z 1387.171,A 0.000,B 0.000,C 90.000,E1 210.797} C_DIS
LIN {X 0.012,Y -141.592,Z 1387.151,A 0.000,B 0.000,C 90.000,E1 207.129} C_DIS
LIN {X 0.059,Y -139.421,Z 1387.115,A 0.000,B 0.000,C 90.000,E1 200.610} C_DIS
LIN {X -0.021,Y -139.146,Z 1387.104,A 0.000,B 0.000,C 90.000,E1 198.779} C_DIS
LIN {X 0.001,Y -138.346,Z 1387.058,A 0.000,B 0.000,C 90.000,E1 190.366} C_DIS
LIN {X -0.013,Y -139.488,Z 1387.006,A 0.000,B 0.000,C 90.000,E1 181.031} C_DIS
LIN {X 0.067,Y -141.092,Z 1386.975,A 0.000,B 0.000,C 90.000,E1 175.412} C_DIS
LIN {X 0.021,Y -142.470,Z 1386.959,A 0.000,B 0.000,C 90.000,E1 172.648} C_DIS
LIN {X -0.030,Y -144.716,Z 1386.934,A 0.000,B 0.000,C 90.000,E1 168.049} C_DIS
LIN {X 0.062,Y -147.316,Z 1386.913,A 0.000,B 0.000,C 90.000,E1 164.338} C_DIS
LIN {X -0.066,Y -150.637,Z 1386.888,A 0.000,B 0.000,C 90.000,E1 159.826} C_DIS
LIN {X 0.010,Y -154.114,Z 1386.868,A 0.000,B 0.000,C 90.000,E1 156.177} C_DIS
LIN {X -0.066,Y -157.539,Z 1386.848,A 0.000,B 0.000,C 90.000,E1 152.615} C_DIS
LIN {X 0.100,Y -161.776,Z 1386.828,A 0.000,B 0.000,C 90.000,E1 148.997} C_DIS
LIN {X -0.017,Y -165.969,Z 1386.808,A 0.000,B 0.000,C 90.000,E1 145.515} C_DIS
LIN {X -0.021,Y -170.963,Z 1386.789,A 0.000,B 0.000,C 90.000,E1 142.029} C_DIS
LIN {X 0.030,Y -175.832,Z 1386.770,A 0.000,B 0.000,C 90.000,E1 138.566} C_DIS
LIN {X 0.025,Y -181.438,Z 1386.751,A 0.000,B 0.000,C 90.000,E1 135.162} C_DIS
LIN {X -0.101,Y -186.944,Z 1386.732,A 0.000,B 0.000,C 90.000,E1 131.838} C_DIS
LIN {X -0.102,Y -190.057,Z 1386.723,A 0.000,B 0.000,C 90.000,E1 130.172} C_DIS
LIN {X -0.088,Y -195.832,Z 1386.705,A 0.000,B 0.000,C 90.000,E1 126.870} C_DIS
LIN {X 0.077,Y -199.342,Z 1386.695,A 0.000,B 0.000,C 90.000,E1 125.025} C_DIS
LIN {X 0.069,Y -309.284,Z 1386.695,A 0.000,B 0.000,C 90.000,E1 125.025} C_DIS
LIN {X -0.030,Y -310.905,Z 1386.695,A 0.000,B 0.000,C 90.000,E1 125.025} C_DIS
LIN {X -0.005,Y -314.996,Z 1386.694,A 0.000,B 0.000,C 90.000,E1 124.865} C_DIS
LIN {X 0.099,Y -317.222,Z 1386.693,A 0.000,B 0.000,C 90.000,E1 124.692} C_DIS
LIN {X -0.032,Y -320.276,Z 1386.691,A 0.000,B 0.000,C 90.000,E1 124.405} C_DIS
LIN {X 0.006,Y -323.861,Z 1386.688,A 0.000,B 0.000,C 90.000,E1 123.833} C_DIS
LIN {X 0.088,Y -325.265,Z 1386.686,A 0.000,B 0.000,C 90.000,E1 123.499} C_DIS
LIN {X -0.099,Y -336.870,Z 1386.669,A 0.000,B 0.000,C 90.000,E1 120.384} C_DIS
LIN {X -0.002,Y -348.691,Z 1386.653,A 0.000,B 0.000,C 90.000,E1 117.590} C_DIS
LIN {X -0.188,Y -361.956,Z 1386.638,A 0.000,B 0.000,C 90.000,E1 114.899} C_DIS
LIN {X -0.087,Y -375.056,Z 1386.625,A 0.000,B 0.000,C 90.000,E1 112.514} C_DIS
LIN {X 0.060,Y -389.479,Z 1386.612,A 0.000,B 0.000,C 90.000,E1 110.174} C_DIS
LIN {X -0.198,Y -405.328,Z 1386.599,A 0.000,B 0.000,C 90.000,E1 107.946} C_DIS
LIN {X -0.071,Y -422.713,Z 1386.587,A 0.000,B 0.000,C 90.000,E1 105.717} C_DIS
LIN {X 0.169,Y -441.735,Z 1386.575,A 0.000,B 0.000,C 90.000,E1 103.536} C_DIS
LIN {X 0.049,Y -461.777,Z 1386.564,A 0.000,B 0.000,C 90.000,E1 101.535} C_DIS
LIN {X 0.150,Y -482.361,Z 1386.554,A 0.000,B 0.000,C 90.000,E1 99.670} C_DIS
LIN {X 0.185,Y -484.580,Z 1386.553,A 0.000,B 0.000,C 90.000,E1 99.443} C_DIS
LIN {X 0.109,Y -486.408,Z 1386.551,A 0.000,B 0.000,C 90.000,E1 99.208} C_DIS
LIN {X 0.031,Y -487.784,Z 1386.550,A 0.000,B 0.000,C 90.000,E1 98.973} C_DIS
LIN {X 0.230,Y -489.548,Z 1386.547,A 0.000,B 0.000,C 90.000,E1 98.454} C_DIS
LIN {X -0.046,Y -490.212,Z 1386.544,A 0.000,B 0.000,C 90.000,E1 97.992} C_DIS
LIN {X 0.176,Y -489.888,Z 1386.542,A 0.000,B 0.000,C 90.000,E1 97.473} C_DIS
LIN {X -0.025,Y -488.529,Z 1386.539,A 0.000,B 0.000,C 90.000,E1 97.004} C_DIS
LIN {X -0.186,Y -487.391,Z 1386.537,A 0.000,B 0.000,C 90.000,E1 96.777} C_DIS
LIN {X 0.029,Y -484.131,Z 1386.535,A 0.000,B 0.000,C 90.000,E1 96.258} C_DIS
LIN {X -0.186,Y -467.681,Z 1386.521,A 0.000,B 0.000,C 90.000,E1 93.784} C_DIS
LIN {X -0.018,Y -457.673,Z 1386.512,A 0.000,B 0.000,C 90.000,E1 92.236} C_DIS
LIN {X 0.058,Y -439.969,Z 1386.497,A 0.000,B 0.000,C 90.000,E1 89.370} C_DIS
LIN {X 0.044,Y -427.919,Z 1386.485,A 0.000,B 0.000,C 90.000,E1 87.249} C_DIS
LIN {X -0.016,Y -418.929,Z 1386.476,A 0.000,B 0.000,C 90.000,E1 85.641} C_DIS
LIN {X -0.122,Y -408.168,Z 1386.465,A 0.000,B 0.000,C 90.000,E1 83.742} C_DIS
LIN {X -0.029,Y -398.967,Z 1386.456,A 0.000,B 0.000,C 90.000,E1 82.064} C_DIS
LIN {X -0.043,Y -387.941,Z 1386.445,A 0.000,B 0.000,C 90.000,E1 80.095} C_DIS
LIN {X 0.213,Y -376.658,Z 1386.434,A 0.000,B 0.000,C 90.000,E1 78.049} C_DIS
LIN {X -0.125,Y -366.888,Z 1386.424,A 0.000,B 0.000,C 90.000,E1 76.353} C_DIS
LIN {X -0.105,Y -357.021,Z 1386.414,A 0.000,B 0.000,C 90.000,E1 74.574} C_DIS
LIN {X 0.194,Y -345.363,Z 1386.402,A 0.000,B 0.000,C 90.000,E1 72.417} C_DIS
LIN {X 0.026,Y -335.309,Z 1386.392,A 0.000,B 0.000,C 90.000,E1 70.604} C_DIS
LIN {X -0.029,Y -320.509,Z 1386.377,A 0.000,B 0.000,C 90.000,E1 67.794} C_DIS
LIN {X -0.086,Y -305.189,Z 1386.359,A 0.000,B 0.000,C 90.000,E1 64.588} C_DIS
LIN {X -0.063,Y -295.507,Z 1386.346,A 0.000,B 0.000,C 90.000,E1 62.281} C_DIS
LIN {X 0.007,Y -285.539,Z 1386.331,A 0.000,B 0.000,C 90.000,E1 59.587} C_DIS
LIN {X 0.017,Y -274.450,Z 1386.312,A 0.000,B 0.000,C 90.000,E1 56.167} C_DIS
LIN {X 0.024,Y -264.216,Z 1386.293,A 0.000,B 0.000,C 90.000,E1 52.683} C_DIS
LIN {X 0.000,Y -254.622,Z 1386.273,A 0.000,B 0.000,C 90.000,E1 49.138} C_DIS
LIN {X -0.025,Y -245.607,Z 1386.253,A 0.000,B 0.000,C 90.000,E1 45.526} C_DIS
LIN {X 0.006,Y -237.385,Z 1386.232,A 0.000,B 0.000,C 90.000,E1 41.838} C_DIS
LIN {X 0.006,Y -230.020,Z 1386.212,A 0.000,B 0.000,C 90.000,E1 38.096} C_DIS
LIN {X -0.099,Y -223.652,Z 1386.191,A 0.000,B 0.000,C 90.000,E1 34.326} C_DIS
LIN {X -0.036,Y -218.142,Z 1386.169,A 0.000,B 0.000,C 90.000,E1 30.463} C_DIS
LIN {X -0.008,Y -213.525,Z 1386.148,A 0.000,B 0.000,C 90.000,E1 26.565} C_DIS
LIN {X 0.010,Y -209.359,Z 1386.121,A 0.000,B 0.000,C 90.000,E1 21.844} C_DIS
LIN {X -0.010,Y -206.396,Z 1386.095,A 0.000,B 0.000,C 90.000,E1 17.094} C_DIS
LIN {X -0.044,Y -204.412,Z 1386.073,A 0.000,B 0.000,C 90.000,E1 13.119} C_DIS
LIN {X 0.005,Y -202.980,Z 1386.055,A 0.000,B 0.000,C 90.000,E1 9.905} C_DIS
LIN {X -0.063,Y -201.370,Z 1386.033,A 0.000,B 0.000,C 90.000,E1 5.910} C_DIS
LIN {X -0.095,Y -200.056,Z 1386.010,A 0.000,B 0.000,C 90.000,E1 1.892} C_DIS
LIN {X -0.101,Y -198.918,Z 1385.984,A 0.000,B 0.000,C 90.000,E1 357.135} C_DIS
LIN {X 0.016,Y -198.607,Z 1385.948,A 0.000,B 0.000,C 90.000,E1 350.622} C_DIS
LIN {X -0.023,Y -200.848,Z 1385.903,A 0.000,B 0.000,C 90.000,E1 342.543} C_DIS
LIN {X -0.042,Y -203.902,Z 1385.876,A 0.000,B 0.000,C 90.000,E1 337.720} C_DIS
LIN {X -0.021,Y -207.634,Z 1385.854,A 0.000,B 0.000,C 90.000,E1 333.717} C_DIS
LIN {X 0.018,Y -212.531,Z 1385.832,A 0.000,B 0.000,C 90.000,E1 329.744} C_DIS
LIN {X -0.071,Y -217.351,Z 1385.814,A 0.000,B 0.000,C 90.000,E1 326.628} C_DIS
LIN {X 0.023,Y -223.013,Z 1385.797,A 0.000,B 0.000,C 90.000,E1 323.497} C_DIS
LIN {X -0.012,Y -229.543,Z 1385.780,A 0.000,B 0.000,C 90.000,E1 320.436} C_DIS
LIN {X 0.027,Y -237.983,Z 1385.761,A 0.000,B 0.000,C 90.000,E1 317.025} C_DIS
LIN {X -0.038,Y -247.392,Z 1385.743,A 0.000,B 0.000,C 90.000,E1 313.704} C_DIS
LIN {X -0.016,Y -255.639,Z 1385.729,A 0.000,B 0.000,C 90.000,E1 311.148} C_DIS
LIN {X 0.056,Y -264.804,Z 1385.715,A 0.000,B 0.000,C 90.000,E1 308.624} C_DIS
LIN {X 0.036,Y -277.931,Z 1385.697,A 0.000,B 0.000,C 90.000,E1 305.471} C_DIS
LIN {X -0.140,Y -286.080,Z 1385.688,A 0.000,B 0.000,C 90.000,E1 303.785} C_DIS
LIN {X -0.106,Y -295.313,Z 1385.678,A 0.000,B 0.000,C 90.000,E1 302.084} C_DIS
LIN {X 0.058,Y -303.522,Z 1385.671,A 0.000,B 0.000,C 90.000,E1 300.718} C_DIS
LIN {X 0.019,Y -312.634,Z 1385.663,A 0.000,B 0.000,C 90.000,E1 299.411} C_DIS
LIN {X 0.174,Y -325.500,Z 1385.654,A 0.000,B 0.000,C 90.000,E1 297.769} C_DIS
LIN {X -0.048,Y -344.182,Z 1385.643,A 0.000,B 0.000,C 90.000,E1 295.720} C_DIS
LIN {X 0.008,Y -357.523,Z 1385.635,A 0.000,B 0.000,C 90.000,E1 294.259} C_DIS
LIN {X 0.005,Y -370.747,Z 1385.627,A 0.000,B 0.000,C 90.000,E1 292.823} C_DIS
LIN {X 0.097,Y -381.034,Z 1385.620,A 0.000,B 0.000,C 90.000,E1 291.663} C_DIS
LIN {X -0.071,Y -391.120,Z 1385.614,A 0.000,B 0.000,C 90.000,E1 290.536} C_DIS
LIN {X 0.161,Y -413.235,Z 1385.600,A 0.000,B 0.000,C 90.000,E1 288.000} C_DIS
LIN {X 0.152,Y -423.001,Z 1385.594,A 0.000,B 0.000,C 90.000,E1 286.913} C_DIS
LIN {X -0.099,Y -429.807,Z 1385.590,A 0.000,B 0.000,C 90.000,E1 286.134} C_DIS
LIN {X 0.001,Y -435.912,Z 1385.585,A 0.000,B 0.000,C 90.000,E1 285.315} C_DIS
LIN {X -0.145,Y -441.242,Z 1385.581,A 0.000,B 0.000,C 90.000,E1 284.537} C_DIS
LIN {X 0.070,Y -445.740,Z 1385.576,A 0.000,B 0.000,C 90.000,E1 283.716} C_DIS
LIN {X 0.002,Y -449.431,Z 1385.572,A 0.000,B 0.000,C 90.000,E1 282.939} C_DIS
LIN {X -0.144,Y -452.323,Z 1385.568,A 0.000,B 0.000,C 90.000,E1 282.175} C_DIS
LIN {X -0.176,Y -453.797,Z 1385.565,A 0.000,B 0.000,C 90.000,E1 281.658} C_DIS
LIN {X -0.104,Y -454.876,Z 1385.562,A 0.000,B 0.000,C 90.000,E1 281.130} C_DIS
LIN {X -0.023,Y -455.575,Z 1385.559,A 0.000,B 0.000,C 90.000,E1 280.602} C_DIS
LIN {X 0.061,Y -455.852,Z 1385.556,A 0.000,B 0.000,C 90.000,E1 280.074} C_DIS
LIN {X 0.070,Y -455.670,Z 1385.553,A 0.000,B 0.000,C 90.000,E1 279.557} C_DIS
LIN {X 0.157,Y -455.074,Z 1385.550,A 0.000,B 0.000,C 90.000,E1 279.029} C_DIS
LIN {X 0.170,Y -453.972,Z 1385.547,A 0.000,B 0.000,C 90.000,E1 278.511} C_DIS
LIN {X 0.181,Y -452.377,Z 1385.545,A 0.000,B 0.000,C 90.000,E1 277.992} C_DIS
LIN {X 0.189,Y -450.193,Z 1385.542,A 0.000,B 0.000,C 90.000,E1 277.473} C_DIS
LIN {X 0.237,Y -447.348,Z 1385.539,A 0.000,B 0.000,C 90.000,E1 276.947} C_DIS
LIN {X 0.212,Y -443.722,Z 1385.536,A 0.000,B 0.000,C 90.000,E1 276.429} C_DIS
LIN {X -0.052,Y -441.627,Z 1385.534,A 0.000,B 0.000,C 90.000,E1 276.201} C_DIS
LIN {X 0.170,Y -439.182,Z 1385.533,A 0.000,B 0.000,C 90.000,E1 275.910} C_DIS
LIN {X 0.104,Y -433.456,Z 1385.530,A 0.000,B 0.000,C 90.000,E1 275.391} C_DIS
LIN {X -0.022,Y -427.152,Z 1385.527,A 0.000,B 0.000,C 90.000,E1 274.935} C_DIS
LIN {X -0.073,Y -420.702,Z 1385.525,A 0.000,B 0.000,C 90.000,E1 274.531} C_DIS
LIN {X -0.170,Y -413.999,Z 1385.523,A 0.000,B 0.000,C 90.000,E1 274.188} C_DIS
LIN {X -0.061,Y -404.124,Z 1385.521,A 0.000,B 0.000,C 90.000,E1 273.726} C_DIS
LIN {X 0.021,Y -394.261,Z 1385.519,A 0.000,B 0.000,C 90.000,E1 273.326} C_DIS
LIN {X 0.066,Y -384.399,Z 1385.517,A 0.000,B 0.000,C 90.000,E1 272.980} C_DIS
LIN {X -0.028,Y -374.152,Z 1385.515,A 0.000,B 0.000,C 90.000,E1 272.694} C_DIS
LIN {X -0.111,Y -363.303,Z 1385.514,A 0.000,B 0.000,C 90.000,E1 272.465} C_DIS
LIN {X 0.147,Y -355.623,Z 1385.513,A 0.000,B 0.000,C 90.000,E1 272.293} C_DIS
LIN {X -0.172,Y -346.498,Z 1385.512,A 0.000,B 0.000,C 90.000,E1 272.236} C_DIS
LIN {X -0.128,Y -332.383,Z 1385.512,A 0.000,B 0.000,C 90.000,E1 272.121} C_DIS
LIN {X 0.044,Y -323.277,Z 1385.511,A 0.000,B 0.000,C 90.000,E1 272.064} C_DIS
LIN {X 0.001,Y -181.252,Z 1385.511,A 0.000,B 0.000,C 90.000,E1 272.064} C_DIS
LIN {X -0.030,Y -181.580,Z 1385.502,A 0.000,B 0.000,C 90.000,E1 270.344} C_DIS
LIN {X -0.054,Y -180.902,Z 1385.474,A 0.000,B 0.000,C 90.000,E1 265.298} C_DIS
LIN {X 0.075,Y -180.236,Z 1385.464,A 0.000,B 0.000,C 90.000,E1 263.571} C_DIS
LIN {X -0.084,Y -178.720,Z 1385.441,A 0.000,B 0.000,C 90.000,E1 259.398} C_DIS
LIN {X -0.017,Y -175.768,Z 1385.413,A 0.000,B 0.000,C 90.000,E1 254.283} C_DIS
LIN {X 0.033,Y -171.952,Z 1385.384,A 0.000,B 0.000,C 90.000,E1 249.135} C_DIS
LIN {X 0.009,Y -171.342,Z 1385.379,A 0.000,B 0.000,C 90.000,E1 248.284} C_DIS
LIN {X -0.013,Y -167.595,Z 1385.355,A 0.000,B 0.000,C 90.000,E1 243.973} C_DIS
LIN {X 0.000,Y -166.235,Z 1385.346,A 0.000,B 0.000,C 90.000,E1 242.231} C_DIS
LIN {X -0.012,Y -162.994,Z 1385.326,A 0.000,B 0.000,C 90.000,E1 238.742} C_DIS
LIN {X 0.035,Y -160.914,Z 1385.312,A 0.000,B 0.000,C 90.000,E1 236.087} C_DIS
LIN {X 0.012,Y -157.677,Z 1385.292,A 0.000,B 0.000,C 90.000,E1 232.557} C_DIS
LIN {X -0.050,Y -155.716,Z 1385.277,A 0.000,B 0.000,C 90.000,E1 229.908} C_DIS
LIN {X 0.005,Y -151.977,Z 1385.252,A 0.000,B 0.000,C 90.000,E1 225.405} C_DIS
LIN {X 0.022,Y -150.220,Z 1385.237,A 0.000,B 0.000,C 90.000,E1 222.690} C_DIS
LIN {X -0.055,Y -146.985,Z 1385.212,A 0.000,B 0.000,C 90.000,E1 218.177} C_DIS
LIN {X 0.054,Y -145.570,Z 1385.197,A 0.000,B 0.000,C 90.000,E1 215.391} C_DIS
LIN {X 0.053,Y -142.960,Z 1385.171,A 0.000,B 0.000,C 90.000,E1 210.797} C_DIS
LIN {X -0.016,Y -141.586,Z 1385.151,A 0.000,B 0.000,C 90.000,E1 207.129} C_DIS
LIN {X 0.031,Y -139.419,Z 1385.115,A 0.000,B 0.000,C 90.000,E1 200.610} C_DIS
LIN {X -0.049,Y -139.144,Z 1385.104,A 0.000,B 0.000,C 90.000,E1 198.779} C_DIS
LIN {X -0.027,Y -138.347,Z 1385.057,A 0.000,B 0.000,C 90.000,E1 190.366} C_DIS
LIN {X -0.041,Y -139.490,Z 1385.006,A 0.000,B 0.000,C 90.000,E1 181.031} C_DIS
LIN {X 0.040,Y -141.097,Z 1384.975,A 0.000,B 0.000,C 90.000,E1 175.412} C_DIS
LIN {X -0.007,Y -142.475,Z 1384.959,A 0.000,B 0.000,C 90.000,E1 172.648} C_DIS
LIN {X -0.060,Y -144.722,Z 1384.933,A 0.000,B 0.000,C 90.000,E1 168.049} C_DIS
LIN {X 0.033,Y -147.324,Z 1384.913,A 0.000,B 0.000,C 90.000,E1 164.338} C_DIS
LIN {X -0.043,Y -150.647,Z 1384.888,A 0.000,B 0.000,C 90.000,E1 159.806} C_DIS
LIN {X -0.019,Y -154.124,Z 1384.868,A 0.000,B 0.000,C 90.000,E1 156.177} C_DIS
LIN {X 0.043,Y -157.550,Z 1384.848,A 0.000,B 0.000,C 90.000,E1 152.564} C_DIS
LIN {X 0.069,Y -161.791,Z 1384.828,A 0.000,B 0.000,C 90.000,E1 148.997} C_DIS
LIN {X -0.049,Y -165.983,Z 1384.808,A 0.000,B 0.000,C 90.000,E1 145.515} C_DIS
LIN {X -0.053,Y -170.979,Z 1384.789,A 0.000,B 0.000,C 90.000,E1 142.029} C_DIS
LIN {X -0.002,Y -175.849,Z 1384.770,A 0.000,B 0.000,C 90.000,E1 138.566} C_DIS
LIN {X -0.008,Y -181.453,Z 1384.751,A 0.000,B 0.000,C 90.000,E1 135.162} C_DIS
LIN {X 0.129,Y -186.963,Z 1384.732,A 0.000,B 0.000,C 90.000,E1 131.757} C_DIS
LIN {X -0.013,Y -190.077,Z 1384.723,A 0.000,B 0.000,C 90.000,E1 130.135} C_DIS
LIN {X -0.122,Y -195.851,Z 1384.705,A 0.000,B 0.000,C 90.000,E1 126.870} C_DIS
LIN {X 0.074,Y -199.344,Z 1384.695,A 0.000,B 0.000,C 90.000,E1 125.025} C_DIS
LIN {X 0.065,Y -310.223,Z 1384.695,A 0.000,B 0.000,C 90.000,E1 125.025} C_DIS
LIN {X -0.084,Y -311.641,Z 1384.694,A 0.000,B 0.000,C 90.000,E1 125.025} C_DIS
LIN {X 0.044,Y -317.388,Z 1384.693,A 0.000,B 0.000,C 90.000,E1 124.692} C_DIS
LIN {X -0.088,Y -320.372,Z 1384.691,A 0.000,B 0.000,C 90.000,E1 124.405} C_DIS
LIN {X -0.097,Y -322.380,Z 1384.689,A 0.000,B 0.000,C 90.000,E1 124.119} C_DIS
LIN {X -0.106,Y -323.948,Z 1384.688,A 0.000,B 0.000,C 90.000,E1 123.833} C_DIS
LIN {X -0.018,Y -325.318,Z 1384.686,A 0.000,B 0.000,C 90.000,E1 123.499} C_DIS
LIN {X 0.090,Y -336.916,Z 1384.669,A 0.000,B 0.000,C 90.000,E1 120.335} C_DIS
LIN {X -0.106,Y -348.746,Z 1384.653,A 0.000,B 0.000,C 90.000,E1 117.590} C_DIS
LIN {X 0.034,Y -362.020,Z 1384.638,A 0.000,B 0.000,C 90.000,E1 114.847} C_DIS
LIN {X 0.153,Y -375.128,Z 1384.625,A 0.000,B 0.000,C 90.000,E1 112.461} C_DIS
LIN {X -0.050,Y -389.561,Z 1384.612,A 0.000,B 0.000,C 90.000,E1 110.174} C_DIS
LIN {X 0.200,Y -405.420,Z 1384.599,A 0.000,B 0.000,C 90.000,E1 107.873} C_DIS
LIN {X 0.221,Y -422.817,Z 1384.587,A 0.000,B 0.000,C 90.000,E1 105.662} C_DIS
LIN {X 0.053,Y -441.849,Z 1384.575,A 0.000,B 0.000,C 90.000,E1 103.536} C_DIS
LIN {X -0.065,Y -461.895,Z 1384.564,A 0.000,B 0.000,C 90.000,E1 101.535} C_DIS
LIN {X 0.041,Y -482.478,Z 1384.554,A 0.000,B 0.000,C 90.000,E1 99.670} C_DIS
LIN {X 0.075,Y -484.631,Z 1384.552,A 0.000,B 0.000,C 90.000,E1 99.443} C_DIS
LIN {X -0.037,Y -486.438,Z 1384.551,A 0.000,B 0.000,C 90.000,E1 99.208} C_DIS
LIN {X -0.150,Y -487.793,Z 1384.550,A 0.000,B 0.000,C 90.000,E1 98.973} C_DIS
LIN {X 0.048,Y -489.483,Z 1384.547,A 0.000,B 0.000,C 90.000,E1 98.454} C_DIS
LIN {X -0.228,Y -490.086,Z 1384.544,A 0.000,B 0.000,C 90.000,E1 97.992} C_DIS
LIN {X 0.057,Y -489.702,Z 1384.542,A 0.000,B 0.000,C 90.000,E1 97.466} C_DIS
LIN {X -0.207,Y -488.275,Z 1384.539,A 0.000,B 0.000,C 90.000,E1 97.004} C_DIS
LIN {X 0.115,Y -487.096,Z 1384.537,A 0.000,B 0.000,C 90.000,E1 96.720} C_DIS
LIN {X 0.212,Y -482.029,Z 1384.533,A 0.000,B 0.000,C 90.000,E1 95.967} C_DIS
LIN {X 0.094,Y -467.293,Z 1384.521,A 0.000,B 0.000,C 90.000,E1 93.726} C_DIS
LIN {X -0.208,Y -457.269,Z 1384.512,A 0.000,B 0.000,C 90.000,E1 92.236} C_DIS
LIN {X -0.137,Y -439.602,Z 1384.496,A 0.000,B 0.000,C 90.000,E1 89.370} C_DIS
LIN {X -0.154,Y -427.597,Z 1384.485,A 0.000,B 0.000,C 90.000,E1 87.249} C_DIS
LIN {X 0.203,Y -418.617,Z 1384.476,A 0.000,B 0.000,C 90.000,E1 85.584} C_DIS
LIN {X 0.019,Y -409.420,Z 1384.467,A 0.000,B 0.000,C 90.000,E1 83.970} C_DIS
LIN {X 0.166,Y -398.680,Z 1384.456,A 0.000,B 0.000,C 90.000,E1 82.008} C_DIS
LIN {X 0.081,Y -389.254,Z 1384.446,A 0.000,B 0.000,C 90.000,E1 80.330} C_DIS
LIN {X -0.036,Y -379.647,Z 1384.437,A 0.000,B 0.000,C 90.000,E1 78.634} C_DIS
LIN {X 0.048,Y -369.927,Z 1384.427,A 0.000,B 0.000,C 90.000,E1 76.881} C_DIS
LIN {X 0.087,Y -358.417,Z 1384.416,A 0.000,B 0.000,C 90.000,E1 74.810} C_DIS
LIN {X -0.028,Y -346.761,Z 1384.404,A 0.000,B 0.000,C 90.000,E1 72.725} C_DIS
LIN {X -0.168,Y -336.708,Z 1384.394,A 0.000,B 0.000,C 90.000,E1 70.913} C_DIS
LIN {X -0.174,Y -321.876,Z 1384.378,A 0.000,B 0.000,C 90.000,E1 68.103} C_DIS
LIN {X 0.094,Y -306.418,Z 1384.360,A 0.000,B 0.000,C 90.000,E1 64.845} C_DIS
LIN {X -0.004,Y -296.615,Z 1384.348,A 0.000,B 0.000,C 90.000,E1 62.564} C_DIS
LIN {X 0.082,Y -286.540,Z 1384.333,A 0.000,B 0.000,C 90.000,E1 59.871} C_DIS
LIN {X -0.017,Y -274.323,Z 1384.312,A 0.000,B 0.000,C 90.000,E1 56.135} C_DIS
LIN {X 0.050,Y -264.141,Z 1384.292,A 0.000,B 0.000,C 90.000,E1 52.637} C_DIS
LIN {X 0.013,Y -254.578,Z 1384.273,A 0.000,B 0.000,C 90.000,E1 49.094} C_DIS
LIN {X -0.027,Y -245.611,Z 1384.253,A 0.000,B 0.000,C 90.000,E1 45.486} C_DIS
LIN {X -0.163,Y -237.405,Z 1384.232,A 0.000,B 0.000,C 90.000,E1 41.838} C_DIS
LIN {X 0.025,Y -230.067,Z 1384.211,A 0.000,B 0.000,C 90.000,E1 38.051} C_DIS
LIN {X -0.071,Y -223.734,Z 1384.190,A 0.000,B 0.000,C 90.000,E1 34.278} C_DIS
LIN {X 0.002,Y -218.263,Z 1384.169,A 0.000,B 0.000,C 90.000,E1 30.413} C_DIS
LIN {X -0.055,Y -213.684,Z 1384.147,A 0.000,B 0.000,C 90.000,E1 26.539} C_DIS
LIN {X -0.124,Y -209.567,Z 1384.121,A 0.000,B 0.000,C 90.000,E1 21.844} C_DIS
LIN {X 0.065,Y -206.647,Z 1384.095,A 0.000,B 0.000,C 90.000,E1 17.040} C_DIS
LIN {X 0.041,Y -204.652,Z 1384.073,A 0.000,B 0.000,C 90.000,E1 13.063} C_DIS
LIN {X -0.071,Y -202.854,Z 1384.050,A 0.000,B 0.000,C 90.000,E1 9.095} C_DIS
LIN {X 0.037,Y -201.325,Z 1384.028,A 0.000,B 0.000,C 90.000,E1 5.049} C_DIS
LIN {X 0.013,Y -200.246,Z 1384.010,A 0.000,B 0.000,C 90.000,E1 1.835} C_DIS
LIN {X -0.098,Y -199.114,Z 1383.984,A 0.000,B 0.000,C 90.000,E1 357.135} C_DIS
LIN {X 0.029,Y -198.788,Z 1383.948,A 0.000,B 0.000,C 90.000,E1 350.622} C_DIS
LIN {X 0.001,Y -201.046,Z 1383.903,A 0.000,B 0.000,C 90.000,E1 342.543} C_DIS
LIN {X -0.009,Y -204.116,Z 1383.876,A 0.000,B 0.000,C 90.000,E1 337.720} C_DIS
LIN {X 0.019,Y -207.843,Z 1383.854,A 0.000,B 0.000,C 90.000,E1 333.717} C_DIS
LIN {X 0.065,Y -212.738,Z 1383.832,A 0.000,B 0.000,C 90.000,E1 329.744} C_DIS
LIN {X -0.017,Y -217.560,Z 1383.815,A 0.000,B 0.000,C 90.000,E1 326.628} C_DIS
LIN {X 0.083,Y -223.204,Z 1383.797,A 0.000,B 0.000,C 90.000,E1 323.497} C_DIS
LIN {X 0.055,Y -229.731,Z 1383.780,A 0.000,B 0.000,C 90.000,E1 320.436} C_DIS
LIN {X -0.073,Y -238.150,Z 1383.761,A 0.000,B 0.000,C 90.000,E1 317.067} C_DIS
LIN {X 0.044,Y -247.540,Z 1383.743,A 0.000,B 0.000,C 90.000,E1 313.704} C_DIS
LIN {X 0.073,Y -255.764,Z 1383.729,A 0.000,B 0.000,C 90.000,E1 311.148} C_DIS
LIN {X -0.057,Y -264.913,Z 1383.715,A 0.000,B 0.000,C 90.000,E1 308.669} C_DIS
LIN {X -0.089,Y -278.027,Z 1383.697,A 0.000,B 0.000,C 90.000,E1 305.518} C_DIS
LIN {X -0.033,Y -286.190,Z 1383.688,A 0.000,B 0.000,C 90.000,E1 303.785} C_DIS
LIN {X 0.006,Y -295.368,Z 1383.678,A 0.000,B 0.000,C 90.000,E1 302.084} C_DIS
LIN {X 0.019,Y -303.570,Z 1383.671,A 0.000,B 0.000,C 90.000,E1 300.747} C_DIS
LIN {X 0.138,Y -312.675,Z 1383.664,A 0.000,B 0.000,C 90.000,E1 299.411} C_DIS
LIN {X -0.061,Y -322.846,Z 1383.656,A 0.000,B 0.000,C 90.000,E1 298.153} C_DIS
LIN {X 0.115,Y -344.094,Z 1383.643,A 0.000,B 0.000,C 90.000,E1 295.720} C_DIS
LIN {X 0.059,Y -357.390,Z 1383.635,A 0.000,B 0.000,C 90.000,E1 294.283} C_DIS
LIN {X -0.231,Y -370.514,Z 1383.627,A 0.000,B 0.000,C 90.000,E1 292.898} C_DIS
LIN {X 0.077,Y -380.707,Z 1383.621,A 0.000,B 0.000,C 90.000,E1 291.716} C_DIS
LIN {X 0.138,Y -390.766,Z 1383.614,A 0.000,B 0.000,C 90.000,E1 290.556} C_DIS
LIN {X 0.005,Y -413.002,Z 1383.600,A 0.000,B 0.000,C 90.000,E1 288.055} C_DIS
LIN {X -0.133,Y -422.802,Z 1383.594,A 0.000,B 0.000,C 90.000,E1 286.985} C_DIS
LIN {X 0.142,Y -429.620,Z 1383.590,A 0.000,B 0.000,C 90.000,E1 286.134} C_DIS
LIN {X -0.180,Y -435.789,Z 1383.585,A 0.000,B 0.000,C 90.000,E1 285.371} C_DIS
LIN {X 0.096,Y -441.168,Z 1383.581,A 0.000,B 0.000,C 90.000,E1 284.537} C_DIS
LIN {X -0.120,Y -445.742,Z 1383.576,A 0.000,B 0.000,C 90.000,E1 283.772} C_DIS
LIN {X 0.146,Y -449.463,Z 1383.572,A 0.000,B 0.000,C 90.000,E1 282.952} C_DIS
LIN {X 0.047,Y -450.569,Z 1383.571,A 0.000,B 0.000,C 90.000,E1 282.703} C_DIS
LIN {X 0.006,Y -452.411,Z 1383.568,A 0.000,B 0.000,C 90.000,E1 282.187} C_DIS
LIN {X 0.071,Y -453.938,Z 1383.565,A 0.000,B 0.000,C 90.000,E1 281.658} C_DIS
LIN {X 0.145,Y -455.064,Z 1383.562,A 0.000,B 0.000,C 90.000,E1 281.130} C_DIS
LIN {X 0.227,Y -455.785,Z 1383.559,A 0.000,B 0.000,C 90.000,E1 280.602} C_DIS
LIN {X -0.217,Y -456.091,Z 1383.556,A 0.000,B 0.000,C 90.000,E1 280.141} C_DIS
LIN {X -0.128,Y -455.983,Z 1383.553,A 0.000,B 0.000,C 90.000,E1 279.613} C_DIS
LIN {X -0.111,Y -455.371,Z 1383.550,A 0.000,B 0.000,C 90.000,E1 279.095} C_DIS
LIN {X -0.024,Y -454.316,Z 1383.548,A 0.000,B 0.000,C 90.000,E1 278.568} C_DIS
LIN {X -0.011,Y -452.775,Z 1383.545,A 0.000,B 0.000,C 90.000,E1 278.049} C_DIS
LIN {X -0.002,Y -450.650,Z 1383.542,A 0.000,B 0.000,C 90.000,E1 277.530} C_DIS
LIN {X 0.055,Y -447.881,Z 1383.539,A 0.000,B 0.000,C 90.000,E1 277.004} C_DIS
LIN {X 0.035,Y -444.414,Z 1383.536,A 0.000,B 0.000,C 90.000,E1 276.486} C_DIS
LIN {X -0.003,Y -439.964,Z 1383.533,A 0.000,B 0.000,C 90.000,E1 275.967} C_DIS
LIN {X 0.162,Y -437.361,Z 1383.532,A 0.000,B 0.000,C 90.000,E1 275.682} C_DIS
LIN {X -0.123,Y -431.518,Z 1383.529,A 0.000,B 0.000,C 90.000,E1 275.220} C_DIS
LIN {X 0.013,Y -425.318,Z 1383.526,A 0.000,B 0.000,C 90.000,E1 274.759} C_DIS
LIN {X 0.097,Y -418.880,Z 1383.524,A 0.000,B 0.000,C 90.000,E1 274.359} C_DIS
LIN {X 0.160,Y -412.216,Z 1383.522,A 0.000,B 0.000,C 90.000,E1 274.012} C_DIS
LIN {X -0.102,Y -402.272,Z 1383.520,A 0.000,B 0.000,C 90.000,E1 273.612} C_DIS
LIN {X 0.051,Y -392.437,Z 1383.518,A 0.000,B 0.000,C 90.000,E1 273.212} C_DIS
LIN {X 0.126,Y -382.330,Z 1383.516,A 0.000,B 0.000,C 90.000,E1 272.865} C_DIS
LIN {X 0.137,Y -371.990,Z 1383.514,A 0.000,B 0.000,C 90.000,E1 272.579} C_DIS
LIN {X 0.123,Y -360.603,Z 1383.513,A 0.000,B 0.000,C 90.000,E1 272.350} C_DIS
LIN {X 0.133,Y -347.994,Z 1383.512,A 0.000,B 0.000,C 90.000,E1 272.178} C_DIS
LIN {X -0.169,Y -334.501,Z 1383.512,A 0.000,B 0.000,C 90.000,E1 272.121} C_DIS
LIN {X -0.039,Y -323.193,Z 1383.511,A 0.000,B 0.000,C 90.000,E1 272.064} C_DIS
LIN {X -0.046,Y -181.254,Z 1383.511,A 0.000,B 0.000,C 90.000,E1 272.064} C_DIS
LIN {X -0.056,Y -181.580,Z 1383.502,A 0.000,B 0.000,C 90.000,E1 270.344} C_DIS
LIN {X -0.080,Y -180.902,Z 1383.474,A 0.000,B 0.000,C 90.000,E1 265.298} C_DIS
LIN {X 0.049,Y -180.232,Z 1383.464,A 0.000,B 0.000,C 90.000,E1 263.571} C_DIS
LIN {X 0.065,Y -178.715,Z 1383.441,A 0.000,B 0.000,C 90.000,E1 259.342} C_DIS
LIN {X -0.042,Y -175.763,Z 1383.413,A 0.000,B 0.000,C 90.000,E1 254.283} C_DIS
LIN {X 0.007,Y -171.947,Z 1383.384,A 0.000,B 0.000,C 90.000,E1 249.135} C_DIS
LIN {X -0.017,Y -171.334,Z 1383.379,A 0.000,B 0.000,C 90.000,E1 248.284} C_DIS
LIN {X 0.036,Y -167.588,Z 1383.355,A 0.000,B 0.000,C 90.000,E1 243.948} C_DIS
LIN {X -0.025,Y -166.227,Z 1383.346,A 0.000,B 0.000,C 90.000,E1 242.231} C_DIS
LIN {X -0.036,Y -162.987,Z 1383.326,A 0.000,B 0.000,C 90.000,E1 238.742} C_DIS
LIN {X 0.011,Y -160.904,Z 1383.312,A 0.000,B 0.000,C 90.000,E1 236.087} C_DIS
LIN {X -0.012,Y -157.670,Z 1383.292,A 0.000,B 0.000,C 90.000,E1 232.557} C_DIS
LIN {X -0.073,Y -155.708,Z 1383.277,A 0.000,B 0.000,C 90.000,E1 229.908} C_DIS
LIN {X -0.018,Y -151.971,Z 1383.252,A 0.000,B 0.000,C 90.000,E1 225.405} C_DIS
LIN {X -0.002,Y -150.213,Z 1383.237,A 0.000,B 0.000,C 90.000,E1 222.690} C_DIS
LIN {X -0.078,Y -146.979,Z 1383.212,A 0.000,B 0.000,C 90.000,E1 218.177} C_DIS
LIN {X 0.031,Y -145.565,Z 1383.197,A 0.000,B 0.000,C 90.000,E1 215.391} C_DIS
LIN {X 0.031,Y -142.956,Z 1383.171,A 0.000,B 0.000,C 90.000,E1 210.797} C_DIS
LIN {X -0.039,Y -141.583,Z 1383.151,A 0.000,B 0.000,C 90.000,E1 207.129} C_DIS
LIN {X 0.008,Y -139.416,Z 1383.115,A 0.000,B 0.000,C 90.000,E1 200.610} C_DIS
LIN {X 0.061,Y -139.141,Z 1383.104,A 0.000,B 0.000,C 90.000,E1 198.725} C_DIS
LIN {X -0.049,Y -138.347,Z 1383.057,A 0.000,B 0.000,C 90.000,E1 190.366} C_DIS
LIN {X -0.064,Y -139.491,Z 1383.006,A 0.000,B 0.000,C 90.000,E1 181.031} C_DIS
LIN {X 0.017,Y -141.101,Z 1382.975,A 0.000,B 0.000,C 90.000,E1 175.412} C_DIS
LIN {X -0.030,Y -142.479,Z 1382.959,A 0.000,B 0.000,C 90.000,E1 172.648} C_DIS
LIN {X 0.058,Y -144.728,Z 1382.933,A 0.000,B 0.000,C 90.000,E1 167.993} C_DIS
LIN {X 0.010,Y -147.332,Z 1382.913,A 0.000,B 0.000,C 90.000,E1 164.338} C_DIS
LIN {X 0.076,Y -150.654,Z 1382.888,A 0.000,B 0.000,C 90.000,E1 159.752} C_DIS
LIN {X -0.044,Y -154.132,Z 1382.868,A 0.000,B 0.000,C 90.000,E1 156.177} C_DIS
LIN {X 0.019,Y -157.561,Z 1382.848,A 0.000,B 0.000,C 90.000,E1 152.564} C_DIS
LIN {X 0.044,Y -161.802,Z 1382.828,A 0.000,B 0.000,C 90.000,E1 148.997} C_DIS
LIN {X 0.063,Y -165.994,Z 1382.808,A 0.000,B 0.000,C 90.000,E1 145.468} C_DIS
LIN {X 0.057,Y -170.991,Z 1382.789,A 0.000,B 0.000,C 90.000,E1 141.984} C_DIS
LIN {X -0.028,Y -175.861,Z 1382.770,A 0.000,B 0.000,C 90.000,E1 138.566} C_DIS
LIN {X -0.035,Y -181.466,Z 1382.751,A 0.000,B 0.000,C 90.000,E1 135.162} C_DIS
LIN {X 0.102,Y -186.978,Z 1382.732,A 0.000,B 0.000,C 90.000,E1 131.757} C_DIS
LIN {X 0.104,Y -190.093,Z 1382.723,A 0.000,B 0.000,C 90.000,E1 130.092} C_DIS
LIN {X 0.008,Y -195.866,Z 1382.705,A 0.000,B 0.000,C 90.000,E1 126.824} C_DIS
LIN {X 0.115,Y -199.320,Z 1382.695,A 0.000,B 0.000,C 90.000,E1 125.025} C_DIS
LIN {X 0.143,Y -309.546,Z 1382.695,A 0.000,B 0.000,C 90.000,E1 125.025} C_DIS
LIN {X -0.127,Y -312.154,Z 1382.694,A 0.000,B 0.000,C 90.000,E1 125.025} C_DIS
LIN {X 0.000,Y -317.526,Z 1382.693,A 0.000,B 0.000,C 90.000,E1 124.692} C_DIS
LIN {X -0.133,Y -320.451,Z 1382.691,A 0.000,B 0.000,C 90.000,E1 124.405} C_DIS
LIN {X 0.101,Y -322.455,Z 1382.689,A 0.000,B 0.000,C 90.000,E1 124.072} C_DIS
LIN {X 0.068,Y -324.020,Z 1382.688,A 0.000,B 0.000,C 90.000,E1 123.785} C_DIS
LIN {X -0.113,Y -325.363,Z 1382.686,A 0.000,B 0.000,C 90.000,E1 123.499} C_DIS
LIN {X -0.007,Y -336.960,Z 1382.669,A 0.000,B 0.000,C 90.000,E1 120.335} C_DIS
LIN {X -0.044,Y -348.798,Z 1382.653,A 0.000,B 0.000,C 90.000,E1 117.564} C_DIS
LIN {X 0.085,Y -362.081,Z 1382.638,A 0.000,B 0.000,C 90.000,E1 114.823} C_DIS
LIN {X 0.049,Y -375.198,Z 1382.625,A 0.000,B 0.000,C 90.000,E1 112.461} C_DIS
LIN {X 0.211,Y -389.640,Z 1382.612,A 0.000,B 0.000,C 90.000,E1 110.120} C_DIS
LIN {X 0.092,Y -405.508,Z 1382.599,A 0.000,B 0.000,C 90.000,E1 107.873} C_DIS
LIN {X 0.112,Y -422.915,Z 1382.587,A 0.000,B 0.000,C 90.000,E1 105.662} C_DIS
LIN {X -0.060,Y -441.958,Z 1382.575,A 0.000,B 0.000,C 90.000,E1 103.536} C_DIS
LIN {X -0.174,Y -462.008,Z 1382.564,A 0.000,B 0.000,C 90.000,E1 101.535} C_DIS
LIN {X -0.064,Y -482.579,Z 1382.554,A 0.000,B 0.000,C 90.000,E1 99.670} C_DIS
LIN {X -0.030,Y -484.666,Z 1382.552,A 0.000,B 0.000,C 90.000,E1 99.443} C_DIS
LIN {X -0.143,Y -486.426,Z 1382.551,A 0.000,B 0.000,C 90.000,E1 99.208} C_DIS
LIN {X 0.224,Y -487.745,Z 1382.550,A 0.000,B 0.000,C 90.000,E1 98.916} C_DIS
LIN {X -0.061,Y -489.383,Z 1382.547,A 0.000,B 0.000,C 90.000,E1 98.454} C_DIS
LIN {X 0.149,Y -489.943,Z 1382.544,A 0.000,B 0.000,C 90.000,E1 97.936} C_DIS
LIN {X -0.053,Y -489.517,Z 1382.542,A 0.000,B 0.000,C 90.000,E1 97.466} C_DIS
LIN {X 0.168,Y -488.041,Z 1382.539,A 0.000,B 0.000,C 90.000,E1 96.947} C_DIS
LIN {X 0.005,Y -486.830,Z 1382.537,A 0.000,B 0.000,C 90.000,E1 96.720} C_DIS
LIN {X -0.022,Y -466.961,Z 1382.521,A 0.000,B 0.000,C 90.000,E1 93.726} C_DIS
LIN {X 0.131,Y -456.914,Z 1382.512,A 0.000,B 0.000,C 90.000,E1 92.178} C_DIS
LIN {X -0.005,Y -440.807,Z 1382.498,A 0.000,B 0.000,C 90.000,E1 89.599} C_DIS
LIN {X 0.004,Y -428.811,Z 1382.486,A 0.000,B 0.000,C 90.000,E1 87.478} C_DIS
LIN {X -0.037,Y -419.882,Z 1382.477,A 0.000,B 0.000,C 90.000,E1 85.869} C_DIS
LIN {X 0.177,Y -410.753,Z 1382.468,A 0.000,B 0.000,C 90.000,E1 84.204} C_DIS
LIN {X -0.051,Y -400.009,Z 1382.457,A 0.000,B 0.000,C 90.000,E1 82.299} C_DIS
LIN {X -0.109,Y -390.623,Z 1382.448,A 0.000,B 0.000,C 90.000,E1 80.622} C_DIS
LIN {X 0.174,Y -381.072,Z 1382.438,A 0.000,B 0.000,C 90.000,E1 78.870} C_DIS
LIN {X -0.086,Y -369.752,Z 1382.427,A 0.000,B 0.000,C 90.000,E1 76.881} C_DIS
LIN {X -0.014,Y -359.891,Z 1382.417,A 0.000,B 0.000,C 90.000,E1 75.102} C_DIS
LIN {X -0.084,Y -348.225,Z 1382.406,A 0.000,B 0.000,C 90.000,E1 73.015} C_DIS
LIN {X 0.130,Y -338.191,Z 1382.395,A 0.000,B 0.000,C 90.000,E1 71.148} C_DIS
LIN {X 0.076,Y -324.911,Z 1382.382,A 0.000,B 0.000,C 90.000,E1 68.666} C_DIS
LIN {X -0.078,Y -307.697,Z 1382.362,A 0.000,B 0.000,C 90.000,E1 65.177} C_DIS
LIN {X 0.002,Y -296.451,Z 1382.347,A 0.000,B 0.000,C 90.000,E1 62.538} C_DIS
LIN {X -0.050,Y -286.393,Z 1382.333,A 0.000,B 0.000,C 90.000,E1 59.871} C_DIS
LIN {X 0.081,Y -274.237,Z 1382.312,A 0.000,B 0.000,C 90.000,E1 56.087} C_DIS
LIN {X -0.062,Y -266.082,Z 1382.296,A 0.000,B 0.000,C 90.000,E1 53.336} C_DIS
LIN {X 0.005,Y -256.429,Z 1382.277,A 0.000,B 0.000,C 90.000,E1 49.784} C_DIS
LIN {X -0.149,Y -247.391,Z 1382.257,A 0.000,B 0.000,C 90.000,E1 46.215} C_DIS
LIN {X -0.066,Y -239.021,Z 1382.236,A 0.000,B 0.000,C 90.000,E1 42.528} C_DIS
LIN {X 0.135,Y -231.552,Z 1382.215,A 0.000,B 0.000,C 90.000,E1 38.749} C_DIS
LIN {X -0.110,Y -225.013,Z 1382.194,A 0.000,B 0.000,C 90.000,E1 35.025} C_DIS
LIN {X 0.116,Y -219.406,Z 1382.173,A 0.000,B 0.000,C 90.000,E1 31.131} C_DIS
LIN {X 0.090,Y -214.668,Z 1382.152,A 0.000,B 0.000,C 90.000,E1 27.257} C_DIS
LIN {X -0.048,Y -210.368,Z 1382.125,A 0.000,B 0.000,C 90.000,E1 22.589} C_DIS
LIN {X -0.009,Y -206.908,Z 1382.095,A 0.000,B 0.000,C 90.000,E1 17.040} C_DIS
LIN {X -0.025,Y -204.877,Z 1382.073,A 0.000,B 0.000,C 90.000,E1 13.063} C_DIS
LIN {X 0.104,Y -203.058,Z 1382.050,A 0.000,B 0.000,C 90.000,E1 9.029} C_DIS
LIN {X -0.014,Y -201.834,Z 1382.032,A 0.000,B 0.000,C 90.000,E1 5.853} C_DIS
LIN {X -0.018,Y -200.704,Z 1382.015,A 0.000,B 0.000,C 90.000,E1 2.636} C_DIS
LIN {X -0.071,Y -199.447,Z 1381.988,A 0.000,B 0.000,C 90.000,E1 357.936} C_DIS
LIN {X 0.039,Y -198.908,Z 1381.953,A 0.000,B 0.000,C 90.000,E1 351.432} C_DIS
LIN {X -0.072,Y -200.866,Z 1381.908,A 0.000,B 0.000,C 90.000,E1 343.378} C_DIS
LIN {X 0.022,Y -204.320,Z 1381.876,A 0.000,B 0.000,C 90.000,E1 337.720} C_DIS
LIN {X 0.058,Y -208.054,Z 1381.854,A 0.000,B 0.000,C 90.000,E1 333.717} C_DIS
LIN {X -0.073,Y -212.943,Z 1381.832,A 0.000,B 0.000,C 90.000,E1 329.793} C_DIS
LIN {X 0.035,Y -217.763,Z 1381.815,A 0.000,B 0.000,C 90.000,E1 326.628} C_DIS
LIN {X -0.038,Y -223.395,Z 1381.797,A 0.000,B 0.000,C 90.000,E1 323.543} C_DIS
LIN {X 0.120,Y -229.916,Z 1381.780,A 0.000,B 0.000,C 90.000,E1 320.436} C_DIS
LIN {X -0.125,Y -237.338,Z 1381.764,A 0.000,B 0.000,C 90.000,E1 317.472} C_DIS
LIN {X -0.042,Y -246.582,Z 1381.745,A 0.000,B 0.000,C 90.000,E1 314.109} C_DIS
LIN {X -0.040,Y -254.654,Z 1381.731,A 0.000,B 0.000,C 90.000,E1 311.553} C_DIS
LIN {X 0.029,Y -265.029,Z 1381.715,A 0.000,B 0.000,C 90.000,E1 308.669} C_DIS
LIN {X 0.004,Y -278.130,Z 1381.697,A 0.000,B 0.000,C 90.000,E1 305.518} C_DIS
LIN {X 0.065,Y -286.297,Z 1381.688,A 0.000,B 0.000,C 90.000,E1 303.785} C_DIS
LIN {X 0.108,Y -295.440,Z 1381.678,A 0.000,B 0.000,C 90.000,E1 302.084} C_DIS
LIN {X -0.136,Y -303.642,Z 1381.671,A 0.000,B 0.000,C 90.000,E1 300.797} C_DIS
LIN {X -0.023,Y -312.747,Z 1381.664,A 0.000,B 0.000,C 90.000,E1 299.461} C_DIS
LIN {X -0.009,Y -322.759,Z 1381.656,A 0.000,B 0.000,C 90.000,E1 298.180} C_DIS
LIN {X -0.044,Y -343.806,Z 1381.643,A 0.000,B 0.000,C 90.000,E1 295.796} C_DIS
LIN {X 0.028,Y -357.109,Z 1381.635,A 0.000,B 0.000,C 90.000,E1 294.335} C_DIS
LIN {X 0.064,Y -370.226,Z 1381.627,A 0.000,B 0.000,C 90.000,E1 292.898} C_DIS
LIN {X -0.063,Y -380.534,Z 1381.621,A 0.000,B 0.000,C 90.000,E1 291.770} C_DIS
LIN {X -0.011,Y -390.572,Z 1381.615,A 0.000,B 0.000,C 90.000,E1 290.610} C_DIS
LIN {X 0.220,Y -412.793,Z 1381.600,A 0.000,B 0.000,C 90.000,E1 288.055} C_DIS
LIN {X 0.083,Y -422.630,Z 1381.594,A 0.000,B 0.000,C 90.000,E1 286.985} C_DIS
LIN {X -0.171,Y -429.451,Z 1381.590,A 0.000,B 0.000,C 90.000,E1 286.205} C_DIS
LIN {X 0.040,Y -435.685,Z 1381.585,A 0.000,B 0.000,C 90.000,E1 285.371} C_DIS
LIN {X -0.109,Y -441.107,Z 1381.581,A 0.000,B 0.000,C 90.000,E1 284.592} C_DIS
LIN {X 0.103,Y -445.746,Z 1381.577,A 0.000,B 0.000,C 90.000,E1 283.772} C_DIS
LIN {X 0.130,Y -448.378,Z 1381.574,A 0.000,B 0.000,C 90.000,E1 283.244} C_DIS
LIN {X 0.175,Y -450.615,Z 1381.571,A 0.000,B 0.000,C 90.000,E1 282.715} C_DIS
LIN {X -0.209,Y -452.503,Z 1381.568,A 0.000,B 0.000,C 90.000,E1 282.243} C_DIS
LIN {X -0.146,Y -454.085,Z 1381.565,A 0.000,B 0.000,C 90.000,E1 281.715} C_DIS
LIN {X -0.072,Y -455.251,Z 1381.562,A 0.000,B 0.000,C 90.000,E1 281.186} C_DIS
LIN {X 0.009,Y -456.018,Z 1381.559,A 0.000,B 0.000,C 90.000,E1 280.658} C_DIS
LIN {X 0.015,Y -456.332,Z 1381.556,A 0.000,B 0.000,C 90.000,E1 280.141} C_DIS
LIN {X 0.106,Y -456.255,Z 1381.553,A 0.000,B 0.000,C 90.000,E1 279.613} C_DIS
LIN {X 0.123,Y -455.698,Z 1381.551,A 0.000,B 0.000,C 90.000,E1 279.095} C_DIS
LIN {X 0.210,Y -454.642,Z 1381.548,A 0.000,B 0.000,C 90.000,E1 278.568} C_DIS
LIN {X -0.224,Y -453.125,Z 1381.545,A 0.000,B 0.000,C 90.000,E1 278.106} C_DIS
LIN {X -0.212,Y -451.060,Z 1381.542,A 0.000,B 0.000,C 90.000,E1 277.587} C_DIS
LIN {X -0.206,Y -448.352,Z 1381.539,A 0.000,B 0.000,C 90.000,E1 277.068} C_DIS
LIN {X -0.168,Y -445.005,Z 1381.536,A 0.000,B 0.000,C 90.000,E1 276.543} C_DIS
LIN {X 0.237,Y -440.710,Z 1381.533,A 0.000,B 0.000,C 90.000,E1 275.967} C_DIS
LIN {X -0.033,Y -438.192,Z 1381.532,A 0.000,B 0.000,C 90.000,E1 275.739} C_DIS
LIN {X 0.101,Y -432.500,Z 1381.529,A 0.000,B 0.000,C 90.000,E1 275.220} C_DIS
LIN {X 0.197,Y -426.351,Z 1381.527,A 0.000,B 0.000,C 90.000,E1 274.759} C_DIS
LIN {X -0.187,Y -419.971,Z 1381.524,A 0.000,B 0.000,C 90.000,E1 274.416} C_DIS
LIN {X -0.179,Y -413.352,Z 1381.522,A 0.000,B 0.000,C 90.000,E1 274.069} C_DIS
LIN {X -0.091,Y -403.360,Z 1381.520,A 0.000,B 0.000,C 90.000,E1 273.612} C_DIS
LIN {X 0.054,Y -393.627,Z 1381.518,A 0.000,B 0.000,C 90.000,E1 273.212} C_DIS
LIN {X 0.083,Y -383.376,Z 1381.516,A 0.000,B 0.000,C 90.000,E1 272.865} C_DIS
LIN {X 0.114,Y -373.246,Z 1381.514,A 0.000,B 0.000,C 90.000,E1 272.579} C_DIS
LIN {X 0.066,Y -361.623,Z 1381.513,A 0.000,B 0.000,C 90.000,E1 272.350} C_DIS
LIN {X 0.070,Y -349.201,Z 1381.512,A 0.000,B 0.000,C 90.000,E1 272.178} C_DIS
LIN {X 0.100,Y -335.498,Z 1381.512,A 0.000,B 0.000,C 90.000,E1 272.064} C_DIS
LIN {X -0.108,Y -324.664,Z 1381.511,A 0.000,B 0.000,C 90.000,E1 272.064} C_DIS
LIN {X -0.086,Y -181.255,Z 1381.511,A 0.000,B 0.000,C 90.000,E1 272.064} C_DIS
LIN {X 0.081,Y -181.581,Z 1381.502,A 0.000,B 0.000,C 90.000,E1 270.286} C_DIS
LIN {X 0.056,Y -180.901,Z 1381.474,A 0.000,B 0.000,C 90.000,E1 265.241} C_DIS
LIN {X 0.005,Y -180.226,Z 1381.464,A 0.000,B 0.000,C 90.000,E1 263.571} C_DIS
LIN {X -0.041,Y -179.039,Z 1381.446,A 0.000,B 0.000,C 90.000,E1 260.208} C_DIS
LIN {X 0.022,Y -178.706,Z 1381.441,A 0.000,B 0.000,C 90.000,E1 259.342} C_DIS
LIN {X -0.037,Y -175.755,Z 1381.412,A 0.000,B 0.000,C 90.000,E1 254.267} C_DIS
LIN {X -0.035,Y -171.939,Z 1381.384,A 0.000,B 0.000,C 90.000,E1 249.135} C_DIS
LIN {X -0.059,Y -171.321,Z 1381.379,A 0.000,B 0.000,C 90.000,E1 248.284} C_DIS
LIN {X -0.005,Y -167.578,Z 1381.355,A 0.000,B 0.000,C 90.000,E1 243.948} C_DIS
LIN {X -0.067,Y -166.212,Z 1381.346,A 0.000,B 0.000,C 90.000,E1 242.231} C_DIS
LIN {X -0.077,Y -162.975,Z 1381.326,A 0.000,B 0.000,C 90.000,E1 238.742} C_DIS
LIN {X -0.030,Y -160.889,Z 1381.312,A 0.000,B 0.000,C 90.000,E1 236.087} C_DIS
LIN {X -0.052,Y -157.659,Z 1381.292,A 0.000,B 0.000,C 90.000,E1 232.557} C_DIS
LIN {X 0.006,Y -155.697,Z 1381.277,A 0.000,B 0.000,C 90.000,E1 229.865} C_DIS
LIN {X -0.058,Y -151.961,Z 1381.252,A 0.000,B 0.000,C 90.000,E1 225.405} C_DIS
LIN {X -0.041,Y -150.201,Z 1381.237,A 0.000,B 0.000,C 90.000,E1 222.690} C_DIS
LIN {X 0.091,Y -146.970,Z 1381.212,A 0.000,B 0.000,C 90.000,E1 218.096} C_DIS
LIN {X -0.007,Y -145.557,Z 1381.197,A 0.000,B 0.000,C 90.000,E1 215.391} C_DIS
LIN {X -0.007,Y -142.950,Z 1381.171,A 0.000,B 0.000,C 90.000,E1 210.797} C_DIS
LIN {X -0.076,Y -141.575,Z 1381.151,A 0.000,B 0.000,C 90.000,E1 207.129} C_DIS
LIN {X -0.029,Y -139.414,Z 1381.114,A 0.000,B 0.000,C 90.000,E1 200.610} C_DIS
LIN {X 0.024,Y -139.138,Z 1381.104,A 0.000,B 0.000,C 90.000,E1 198.725} C_DIS
LIN {X 0.050,Y -138.349,Z 1381.057,A 0.000,B 0.000,C 90.000,E1 190.310} C_DIS
LIN {X 0.038,Y -139.494,Z 1381.005,A 0.000,B 0.000,C 90.000,E1 180.974} C_DIS
LIN {X -0.021,Y -141.107,Z 1380.974,A 0.000,B 0.000,C 90.000,E1 175.412} C_DIS
LIN {X -0.067,Y -142.486,Z 1380.959,A 0.000,B 0.000,C 90.000,E1 172.648} C_DIS
LIN {X 0.021,Y -144.737,Z 1380.933,A 0.000,B 0.000,C 90.000,E1 167.993} C_DIS
LIN {X -0.029,Y -147.343,Z 1380.913,A 0.000,B 0.000,C 90.000,E1 164.338} C_DIS
LIN {X 0.035,Y -150.667,Z 1380.888,A 0.000,B 0.000,C 90.000,E1 159.752} C_DIS
LIN {X -0.084,Y -154.146,Z 1380.867,A 0.000,B 0.000,C 90.000,E1 156.177} C_DIS
LIN {X 0.051,Y -157.576,Z 1380.848,A 0.000,B 0.000,C 90.000,E1 152.538} C_DIS
LIN {X 0.003,Y -161.821,Z 1380.828,A 0.000,B 0.000,C 90.000,E1 148.997} C_DIS
LIN {X 0.022,Y -166.012,Z 1380.808,A 0.000,B 0.000,C 90.000,E1 145.468} C_DIS
LIN {X 0.014,Y -171.013,Z 1380.789,A 0.000,B 0.000,C 90.000,E1 141.984} C_DIS
LIN {X 0.046,Y -175.883,Z 1380.770,A 0.000,B 0.000,C 90.000,E1 138.528} C_DIS
LIN {X -0.079,Y -181.487,Z 1380.751,A 0.000,B 0.000,C 90.000,E1 135.162} C_DIS
LIN {X 0.058,Y -187.002,Z 1380.732,A 0.000,B 0.000,C 90.000,E1 131.757} C_DIS
LIN {X 0.060,Y -190.120,Z 1380.723,A 0.000,B 0.000,C 90.000,E1 130.092} C_DIS
LIN {X 0.079,Y -195.891,Z 1380.704,A 0.000,B 0.000,C 90.000,E1 126.790} C_DIS
LIN {X -0.121,Y -199.295,Z 1380.695,A 0.000,B 0.000,C 90.000,E1 125.105} C_DIS
LIN {X 0.192,Y -309.202,Z 1380.695,A 0.000,B 0.000,C 90.000,E1 125.025} C_DIS
LIN {X 0.142,Y -310.233,Z 1380.695,A 0.000,B 0.000,C 90.000,E1 125.025} C_DIS
LIN {X -0.098,Y -314.977,Z 1380.694,A 0.000,B 0.000,C 90.000,E1 124.898} C_DIS
LIN {X 0.100,Y -317.356,Z 1380.693,A 0.000,B 0.000,C 90.000,E1 124.692} C_DIS
LIN {X -0.208,Y -320.566,Z 1380.691,A 0.000,B 0.000,C 90.000,E1 124.405} C_DIS
LIN {X 0.021,Y -322.537,Z 1380.689,A 0.000,B 0.000,C 90.000,E1 124.072} C_DIS
LIN {X -0.016,Y -324.079,Z 1380.688,A 0.000,B 0.000,C 90.000,E1 123.785} C_DIS
LIN {X -0.107,Y -326.501,Z 1380.684,A 0.000,B 0.000,C 90.000,E1 123.166} C_DIS
LIN {X -0.093,Y -336.997,Z 1380.668,A 0.000,B 0.000,C 90.000,E1 120.335} C_DIS
LIN {X 0.179,Y -348.842,Z 1380.653,A 0.000,B 0.000,C 90.000,E1 117.513} C_DIS
LIN {X -0.005,Y -362.132,Z 1380.638,A 0.000,B 0.000,C 90.000,E1 114.823} C_DIS
LIN {X -0.043,Y -375.256,Z 1380.625,A 0.000,B 0.000,C 90.000,E1 112.461} C_DIS
LIN {X 0.116,Y -389.706,Z 1380.612,A 0.000,B 0.000,C 90.000,E1 110.120} C_DIS
LIN {X -0.004,Y -405.584,Z 1380.599,A 0.000,B 0.000,C 90.000,E1 107.873} C_DIS
LIN {X 0.013,Y -422.999,Z 1380.587,A 0.000,B 0.000,C 90.000,E1 105.662} C_DIS
LIN {X -0.159,Y -442.051,Z 1380.575,A 0.000,B 0.000,C 90.000,E1 103.536} C_DIS
LIN {X 0.183,Y -462.106,Z 1380.564,A 0.000,B 0.000,C 90.000,E1 101.478} C_DIS
LIN {X -0.159,Y -482.657,Z 1380.554,A 0.000,B 0.000,C 90.000,E1 99.670} C_DIS
LIN {X -0.123,Y -484.688,Z 1380.552,A 0.000,B 0.000,C 90.000,E1 99.443} C_DIS
LIN {X -0.236,Y -486.406,Z 1380.551,A 0.000,B 0.000,C 90.000,E1 99.208} C_DIS
LIN {X 0.131,Y -487.693,Z 1380.550,A 0.000,B 0.000,C 90.000,E1 98.916} C_DIS
LIN {X -0.155,Y -489.280,Z 1380.547,A 0.000,B 0.000,C 90.000,E1 98.454} C_DIS
LIN {X 0.055,Y -489.797,Z 1380.544,A 0.000,B 0.000,C 90.000,E1 97.936} C_DIS
LIN {X -0.147,Y -489.328,Z 1380.541,A 0.000,B 0.000,C 90.000,E1 97.466} C_DIS
LIN {X 0.072,Y -487.803,Z 1380.539,A 0.000,B 0.000,C 90.000,E1 96.947} C_DIS
LIN {X -0.090,Y -486.562,Z 1380.537,A 0.000,B 0.000,C 90.000,E1 96.720} C_DIS
LIN {X -0.232,Y -469.851,Z 1380.523,A 0.000,B 0.000,C 90.000,E1 94.245} C_DIS
LIN {X 0.217,Y -461.674,Z 1380.516,A 0.000,B 0.000,C 90.000,E1 92.922} C_DIS
LIN {X 0.202,Y -445.156,Z 1380.502,A 0.000,B 0.000,C 90.000,E1 90.344} C_DIS
LIN {X 0.177,Y -430.050,Z 1380.487,A 0.000,B 0.000,C 90.000,E1 87.707} C_DIS
LIN {X -0.154,Y -419.631,Z 1380.477,A 0.000,B 0.000,C 90.000,E1 85.869} C_DIS
LIN {X 0.059,Y -410.527,Z 1380.468,A 0.000,B 0.000,C 90.000,E1 84.204} C_DIS
LIN {X -0.171,Y -399.780,Z 1380.457,A 0.000,B 0.000,C 90.000,E1 82.299} C_DIS
LIN {X 0.155,Y -390.425,Z 1380.448,A 0.000,B 0.000,C 90.000,E1 80.566} C_DIS
LIN {X 0.052,Y -380.870,Z 1380.438,A 0.000,B 0.000,C 90.000,E1 78.870} C_DIS
LIN {X 0.156,Y -371.186,Z 1380.429,A 0.000,B 0.000,C 90.000,E1 77.117} C_DIS
LIN {X -0.194,Y -361.375,Z 1380.419,A 0.000,B 0.000,C 90.000,E1 75.408} C_DIS
LIN {X 0.163,Y -351.384,Z 1380.409,A 0.000,B 0.000,C 90.000,E1 73.559} C_DIS
LIN {X -0.005,Y -341.344,Z 1380.399,A 0.000,B 0.000,C 90.000,E1 71.764} C_DIS
LIN {X 0.135,Y -328.013,Z 1380.385,A 0.000,B 0.000,C 90.000,E1 69.263} C_DIS
LIN {X -0.032,Y -310.496,Z 1380.365,A 0.000,B 0.000,C 90.000,E1 65.793} C_DIS
LIN {X -0.014,Y -298.985,Z 1380.351,A 0.000,B 0.000,C 90.000,E1 63.179} C_DIS
LIN {X 0.001,Y -288.655,Z 1380.336,A 0.000,B 0.000,C 90.000,E1 60.511} C_DIS
LIN {X 0.045,Y -279.475,Z 1380.321,A 0.000,B 0.000,C 90.000,E1 57.788} C_DIS
LIN {X 0.024,Y -270.057,Z 1380.304,A 0.000,B 0.000,C 90.000,E1 54.689} C_DIS
LIN {X -0.062,Y -262.112,Z 1380.288,A 0.000,B 0.000,C 90.000,E1 51.904} C_DIS
LIN {X 0.008,Y -252.755,Z 1380.268,A 0.000,B 0.000,C 90.000,E1 48.324} C_DIS
LIN {X 0.092,Y -245.676,Z 1380.252,A 0.000,B 0.000,C 90.000,E1 45.405} C_DIS
LIN {X -0.048,Y -237.508,Z 1380.232,A 0.000,B 0.000,C 90.000,E1 41.757} C_DIS
LIN {X -0.043,Y -230.232,Z 1380.211,A 0.000,B 0.000,C 90.000,E1 38.016} C_DIS
LIN {X 0.042,Y -223.943,Z 1380.190,A 0.000,B 0.000,C 90.000,E1 34.199} C_DIS
LIN {X -0.073,Y -218.512,Z 1380.169,A 0.000,B 0.000,C 90.000,E1 30.384} C_DIS
LIN {X -0.038,Y -214.008,Z 1380.147,A 0.000,B 0.000,C 90.000,E1 26.488} C_DIS
LIN {X -0.008,Y -209.993,Z 1380.121,A 0.000,B 0.000,C 90.000,E1 21.770} C_DIS
LIN {X -0.075,Y -207.137,Z 1380.095,A 0.000,B 0.000,C 90.000,E1 17.040} C_DIS
LIN {X 0.035,Y -205.504,Z 1380.077,A 0.000,B 0.000,C 90.000,E1 13.828} C_DIS
LIN {X -0.013,Y -203.618,Z 1380.055,A 0.000,B 0.000,C 90.000,E1 9.849} C_DIS
LIN {X -0.059,Y -202.039,Z 1380.032,A 0.000,B 0.000,C 90.000,E1 5.853} C_DIS
LIN {X -0.071,Y -200.601,Z 1380.010,A 0.000,B 0.000,C 90.000,E1 1.835} C_DIS
LIN {X -0.091,Y -199.469,Z 1379.984,A 0.000,B 0.000,C 90.000,E1 357.135} C_DIS
LIN {X 0.053,Y -199.136,Z 1379.948,A 0.000,B 0.000,C 90.000,E1 350.622} C_DIS
LIN {X 0.047,Y -201.436,Z 1379.903,A 0.000,B 0.000,C 90.000,E1 342.543} C_DIS
LIN {X 0.053,Y -204.506,Z 1379.876,A 0.000,B 0.000,C 90.000,E1 337.720} C_DIS
LIN {X -0.091,Y -208.253,Z 1379.854,A 0.000,B 0.000,C 90.000,E1 333.768} C_DIS
LIN {X -0.028,Y -213.141,Z 1379.832,A 0.000,B 0.000,C 90.000,E1 329.793} C_DIS
LIN {X 0.085,Y -217.962,Z 1379.815,A 0.000,B 0.000,C 90.000,E1 326.628} C_DIS
LIN {X 0.056,Y -225.124,Z 1379.793,A 0.000,B 0.000,C 90.000,E1 322.763} C_DIS
LIN {X -0.100,Y -231.875,Z 1379.776,A 0.000,B 0.000,C 90.000,E1 319.747} C_DIS
LIN {X -0.003,Y -240.487,Z 1379.757,A 0.000,B 0.000,C 90.000,E1 316.338} C_DIS
LIN {X 0.014,Y -250.065,Z 1379.739,A 0.000,B 0.000,C 90.000,E1 313.014} C_DIS
LIN {X 0.101,Y -258.526,Z 1379.725,A 0.000,B 0.000,C 90.000,E1 310.458} C_DIS
LIN {X -0.069,Y -269.343,Z 1379.709,A 0.000,B 0.000,C 90.000,E1 307.649} C_DIS
LIN {X 0.038,Y -279.789,Z 1379.696,A 0.000,B 0.000,C 90.000,E1 305.185} C_DIS
LIN {X -0.105,Y -288.135,Z 1379.686,A 0.000,B 0.000,C 90.000,E1 303.499} C_DIS
LIN {X -0.044,Y -297.474,Z 1379.677,A 0.000,B 0.000,C 90.000,E1 301.799} C_DIS
LIN {X -0.010,Y -305.901,Z 1379.669,A 0.000,B 0.000,C 90.000,E1 300.463} C_DIS
LIN {X -0.019,Y -315.234,Z 1379.662,A 0.000,B 0.000,C 90.000,E1 299.155} C_DIS
LIN {X 0.138,Y -330.588,Z 1379.652,A 0.000,B 0.000,C 90.000,E1 297.257} C_DIS
LIN {X -0.027,Y -346.273,Z 1379.642,A 0.000,B 0.000,C 90.000,E1 295.540} C_DIS
LIN {X 0.024,Y -359.634,Z 1379.634,A 0.000,B 0.000,C 90.000,E1 294.079} C_DIS
LIN {X -0.003,Y -372.762,Z 1379.626,A 0.000,B 0.000,C 90.000,E1 292.642} C_DIS
LIN {X 0.055,Y -383.044,Z 1379.619,A 0.000,B 0.000,C 90.000,E1 291.482} C_DIS
LIN {X -0.089,Y -392.964,Z 1379.613,A 0.000,B 0.000,C 90.000,E1 290.355} C_DIS
LIN {X -0.090,Y -412.761,Z 1379.601,A 0.000,B 0.000,C 90.000,E1 288.109} C_DIS
LIN {X 0.135,Y -422.646,Z 1379.594,A 0.000,B 0.000,C 90.000,E1 286.985} C_DIS
LIN {X -0.119,Y -429.493,Z 1379.590,A 0.000,B 0.000,C 90.000,E1 286.205} C_DIS
LIN {X 0.093,Y -435.720,Z 1379.585,A 0.000,B 0.000,C 90.000,E1 285.371} C_DIS
LIN {X -0.055,Y -441.192,Z 1379.581,A 0.000,B 0.000,C 90.000,E1 284.592} C_DIS
LIN {X 0.159,Y -445.850,Z 1379.577,A 0.000,B 0.000,C 90.000,E1 283.772} C_DIS
LIN {X 0.186,Y -448.486,Z 1379.574,A 0.000,B 0.000,C 90.000,E1 283.244} C_DIS
LIN {X -0.208,Y -450.747,Z 1379.571,A 0.000,B 0.000,C 90.000,E1 282.771} C_DIS
LIN {X -0.151,Y -452.694,Z 1379.568,A 0.000,B 0.000,C 90.000,E1 282.243} C_DIS
LIN {X -0.087,Y -454.285,Z 1379.565,A 0.000,B 0.000,C 90.000,E1 281.715} C_DIS
LIN {X -0.012,Y -455.457,Z 1379.562,A 0.000,B 0.000,C 90.000,E1 281.186} C_DIS
LIN {X 0.071,Y -456.253,Z 1379.559,A 0.000,B 0.000,C 90.000,E1 280.658} C_DIS
LIN {X 0.078,Y -456.611,Z 1379.556,A 0.000,B 0.000,C 90.000,E1 280.141} C_DIS
LIN {X 0.171,Y -456.515,Z 1379.553,A 0.000,B 0.000,C 90.000,E1 279.613} C_DIS
LIN {X 0.189,Y -455.951,Z 1379.551,A 0.000,B 0.000,C 90.000,E1 279.095} C_DIS
LIN {X -0.172,Y -454.946,Z 1379.548,A 0.000,B 0.000,C 90.000,E1 278.624} C_DIS
LIN {X -0.155,Y -453.458,Z 1379.545,A 0.000,B 0.000,C 90.000,E1 278.106} C_DIS
LIN {X -0.142,Y -451.422,Z 1379.542,A 0.000,B 0.000,C 90.000,E1 277.587} C_DIS
LIN {X -0.135,Y -448.744,Z 1379.539,A 0.000,B 0.000,C 90.000,E1 277.068} C_DIS
LIN {X 0.107,Y -447.234,Z 1379.538,A 0.000,B 0.000,C 90.000,E1 276.777} C_DIS
LIN {X 0.085,Y -443.459,Z 1379.535,A 0.000,B 0.000,C 90.000,E1 276.258} C_DIS
LIN {X 0.043,Y -438.767,Z 1379.532,A 0.000,B 0.000,C 90.000,E1 275.739} C_DIS
LIN {X 0.157,Y -433.167,Z 1379.529,A 0.000,B 0.000,C 90.000,E1 275.220} C_DIS
LIN {X 0.216,Y -427.005,Z 1379.527,A 0.000,B 0.000,C 90.000,E1 274.759} C_DIS
LIN {X 0.193,Y -420.662,Z 1379.524,A 0.000,B 0.000,C 90.000,E1 274.359} C_DIS
LIN {X 0.132,Y -413.953,Z 1379.522,A 0.000,B 0.000,C 90.000,E1 274.012} C_DIS
LIN {X 0.140,Y -403.845,Z 1379.520,A 0.000,B 0.000,C 90.000,E1 273.555} C_DIS
LIN {X -0.141,Y -394.021,Z 1379.518,A 0.000,B 0.000,C 90.000,E1 273.212} C_DIS
LIN {X -0.110,Y -383.795,Z 1379.516,A 0.000,B 0.000,C 90.000,E1 272.865} C_DIS
LIN {X -0.093,Y -373.299,Z 1379.514,A 0.000,B 0.000,C 90.000,E1 272.579} C_DIS
LIN {X -0.017,Y -365.684,Z 1379.513,A 0.000,B 0.000,C 90.000,E1 272.407} C_DIS
LIN {X -0.124,Y -353.337,Z 1379.512,A 0.000,B 0.000,C 90.000,E1 272.236} C_DIS
LIN {X -0.022,Y -343.331,Z 1379.512,A 0.000,B 0.000,C 90.000,E1 272.121} C_DIS
LIN {X -0.029,Y -334.916,Z 1379.511,A 0.000,B 0.000,C 90.000,E1 272.064} C_DIS
LIN {X 0.143,Y -326.045,Z 1379.511,A 0.000,B 0.000,C 90.000,E1 272.007} C_DIS
LIN {X 0.056,Y -181.258,Z 1379.511,A 0.000,B 0.000,C 90.000,E1 272.007} C_DIS
LIN {X 0.025,Y -181.580,Z 1379.502,A 0.000,B 0.000,C 90.000,E1 270.286} C_DIS
LIN {X 0.000,Y -180.900,Z 1379.474,A 0.000,B 0.000,C 90.000,E1 265.241} C_DIS
LIN {X -0.051,Y -180.218,Z 1379.464,A 0.000,B 0.000,C 90.000,E1 263.571} C_DIS
LIN {X 0.079,Y -179.035,Z 1379.445,A 0.000,B 0.000,C 90.000,E1 260.151} C_DIS
LIN {X -0.034,Y -178.695,Z 1379.441,A 0.000,B 0.000,C 90.000,E1 259.342} C_DIS
LIN {X 0.076,Y -175.744,Z 1379.412,A 0.000,B 0.000,C 90.000,E1 254.212} C_DIS
LIN {X 0.071,Y -171.928,Z 1379.384,A 0.000,B 0.000,C 90.000,E1 249.082} C_DIS
LIN {X 0.046,Y -171.304,Z 1379.379,A 0.000,B 0.000,C 90.000,E1 248.230} C_DIS
LIN {X 0.091,Y -167.565,Z 1379.355,A 0.000,B 0.000,C 90.000,E1 243.896} C_DIS
LIN {X 0.104,Y -166.192,Z 1379.345,A 0.000,B 0.000,C 90.000,E1 242.153} C_DIS
LIN {X 0.093,Y -162.961,Z 1379.326,A 0.000,B 0.000,C 90.000,E1 238.663} C_DIS
LIN {X -0.082,Y -160.870,Z 1379.311,A 0.000,B 0.000,C 90.000,E1 236.087} C_DIS
LIN {X -0.104,Y -157.644,Z 1379.292,A 0.000,B 0.000,C 90.000,E1 232.557} C_DIS
LIN {X 0.055,Y -155.681,Z 1379.277,A 0.000,B 0.000,C 90.000,E1 229.828} C_DIS
LIN {X 0.000,Y -151.947,Z 1379.252,A 0.000,B 0.000,C 90.000,E1 225.364} C_DIS
LIN {X -0.091,Y -150.185,Z 1379.237,A 0.000,B 0.000,C 90.000,E1 222.690} C_DIS
LIN {X 0.040,Y -146.958,Z 1379.212,A 0.000,B 0.000,C 90.000,E1 218.096} C_DIS
LIN {X -0.056,Y -145.546,Z 1379.197,A 0.000,B 0.000,C 90.000,E1 215.391} C_DIS
LIN {X -0.056,Y -142.940,Z 1379.171,A 0.000,B 0.000,C 90.000,E1 210.797} C_DIS
LIN {X 0.001,Y -141.565,Z 1379.150,A 0.000,B 0.000,C 90.000,E1 207.078} C_DIS
LIN {X 0.053,Y -139.410,Z 1379.114,A 0.000,B 0.000,C 90.000,E1 200.556} C_DIS
LIN {X -0.025,Y -139.132,Z 1379.104,A 0.000,B 0.000,C 90.000,E1 198.725} C_DIS
LIN {X 0.002,Y -138.350,Z 1379.057,A 0.000,B 0.000,C 90.000,E1 190.310} C_DIS
LIN {X -0.010,Y -139.496,Z 1379.005,A 0.000,B 0.000,C 90.000,E1 180.974} C_DIS
LIN {X -0.069,Y -141.116,Z 1378.974,A 0.000,B 0.000,C 90.000,E1 175.412} C_DIS
LIN {X 0.025,Y -142.496,Z 1378.959,A 0.000,B 0.000,C 90.000,E1 172.591} C_DIS
LIN {X -0.029,Y -144.749,Z 1378.933,A 0.000,B 0.000,C 90.000,E1 167.993} C_DIS
LIN {X -0.079,Y -147.358,Z 1378.913,A 0.000,B 0.000,C 90.000,E1 164.338} C_DIS
LIN {X -0.015,Y -150.683,Z 1378.887,A 0.000,B 0.000,C 90.000,E1 159.752} C_DIS
LIN {X 0.068,Y -154.164,Z 1378.867,A 0.000,B 0.000,C 90.000,E1 156.102} C_DIS
LIN {X -0.001,Y -157.596,Z 1378.847,A 0.000,B 0.000,C 90.000,E1 152.538} C_DIS
LIN {X -0.050,Y -161.846,Z 1378.828,A 0.000,B 0.000,C 90.000,E1 148.997} C_DIS
LIN {X -0.033,Y -166.037,Z 1378.808,A 0.000,B 0.000,C 90.000,E1 145.468} C_DIS
LIN {X -0.041,Y -171.040,Z 1378.789,A 0.000,B 0.000,C 90.000,E1 141.984} C_DIS
LIN {X -0.011,Y -175.911,Z 1378.770,A 0.000,B 0.000,C 90.000,E1 138.528} C_DIS
LIN {X -0.018,Y -180.148,Z 1378.755,A 0.000,B 0.000,C 90.000,E1 135.972} C_DIS
LIN {X -0.049,Y -185.566,Z 1378.737,A 0.000,B 0.000,C 90.000,E1 132.609} C_DIS
LIN {X 0.001,Y -190.154,Z 1378.723,A 0.000,B 0.000,C 90.000,E1 130.092} C_DIS
LIN {X 0.020,Y -195.923,Z 1378.704,A 0.000,B 0.000,C 90.000,E1 126.790} C_DIS
LIN {X -0.115,Y -199.292,Z 1378.695,A 0.000,B 0.000,C 90.000,E1 125.105} C_DIS
LIN {X 0.201,Y -309.856,Z 1378.695,A 0.000,B 0.000,C 90.000,E1 125.025} C_DIS
LIN {X 0.049,Y -311.430,Z 1378.695,A 0.000,B 0.000,C 90.000,E1 125.025} C_DIS
LIN {X -0.012,Y -315.331,Z 1378.694,A 0.000,B 0.000,C 90.000,E1 124.865} C_DIS
LIN {X 0.005,Y -317.592,Z 1378.693,A 0.000,B 0.000,C 90.000,E1 124.692} C_DIS
LIN {X 0.142,Y -320.706,Z 1378.691,A 0.000,B 0.000,C 90.000,E1 124.326} C_DIS
LIN {X 0.068,Y -322.672,Z 1378.689,A 0.000,B 0.000,C 90.000,E1 124.040} C_DIS
LIN {X -0.187,Y -324.206,Z 1378.688,A 0.000,B 0.000,C 90.000,E1 123.785} C_DIS
LIN {X 0.174,Y -326.584,Z 1378.684,A 0.000,B 0.000,C 90.000,E1 123.086} C_DIS
LIN {X 0.024,Y -337.094,Z 1378.668,A 0.000,B 0.000,C 90.000,E1 120.285} C_DIS
LIN {X 0.000,Y -348.953,Z 1378.653,A 0.000,B 0.000,C 90.000,E1 117.513} C_DIS
LIN {X 0.143,Y -362.259,Z 1378.638,A 0.000,B 0.000,C 90.000,E1 114.771} C_DIS
LIN {X 0.120,Y -375.397,Z 1378.625,A 0.000,B 0.000,C 90.000,E1 112.408} C_DIS
LIN {X -0.072,Y -389.864,Z 1378.612,A 0.000,B 0.000,C 90.000,E1 110.120} C_DIS
LIN {X 0.190,Y -405.759,Z 1378.599,A 0.000,B 0.000,C 90.000,E1 107.819} C_DIS
LIN {X -0.183,Y -423.194,Z 1378.587,A 0.000,B 0.000,C 90.000,E1 105.662} C_DIS
LIN {X 0.072,Y -442.265,Z 1378.575,A 0.000,B 0.000,C 90.000,E1 103.480} C_DIS
LIN {X -0.008,Y -462.326,Z 1378.564,A 0.000,B 0.000,C 90.000,E1 101.478} C_DIS
LIN {X 0.133,Y -482.840,Z 1378.553,A 0.000,B 0.000,C 90.000,E1 99.613} C_DIS
LIN {X 0.252,Y -484.789,Z 1378.552,A 0.000,B 0.000,C 90.000,E1 99.378} C_DIS
LIN {X 0.061,Y -486.444,Z 1378.551,A 0.000,B 0.000,C 90.000,E1 99.151} C_DIS
LIN {X -0.053,Y -487.684,Z 1378.549,A 0.000,B 0.000,C 90.000,E1 98.916} C_DIS
LIN {X 0.146,Y -489.197,Z 1378.547,A 0.000,B 0.000,C 90.000,E1 98.398} C_DIS
LIN {X -0.129,Y -489.651,Z 1378.544,A 0.000,B 0.000,C 90.000,E1 97.936} C_DIS
LIN {X 0.153,Y -489.122,Z 1378.541,A 0.000,B 0.000,C 90.000,E1 97.409} C_DIS
LIN {X -0.113,Y -487.524,Z 1378.539,A 0.000,B 0.000,C 90.000,E1 96.947} C_DIS
LIN {X 0.208,Y -486.236,Z 1378.537,A 0.000,B 0.000,C 90.000,E1 96.663} C_DIS
LIN {X -0.040,Y -472.684,Z 1378.526,A 0.000,B 0.000,C 90.000,E1 94.702} C_DIS
LIN {X 0.209,Y -462.961,Z 1378.518,A 0.000,B 0.000,C 90.000,E1 93.154} C_DIS
LIN {X 0.007,Y -444.769,Z 1378.502,A 0.000,B 0.000,C 90.000,E1 90.344} C_DIS
LIN {X -0.022,Y -429.716,Z 1378.487,A 0.000,B 0.000,C 90.000,E1 87.707} C_DIS
LIN {X 0.065,Y -419.308,Z 1378.477,A 0.000,B 0.000,C 90.000,E1 85.812} C_DIS
LIN {X -0.142,Y -410.220,Z 1378.468,A 0.000,B 0.000,C 90.000,E1 84.204} C_DIS
LIN {X -0.067,Y -401.034,Z 1378.458,A 0.000,B 0.000,C 90.000,E1 82.534} C_DIS
LIN {X 0.016,Y -390.144,Z 1378.448,A 0.000,B 0.000,C 90.000,E1 80.557} C_DIS
LIN {X 0.188,Y -382.190,Z 1378.440,A 0.000,B 0.000,C 90.000,E1 79.106} C_DIS
LIN {X -0.053,Y -372.561,Z 1378.430,A 0.000,B 0.000,C 90.000,E1 77.409} C_DIS
LIN {X -0.020,Y -362.771,Z 1378.420,A 0.000,B 0.000,C 90.000,E1 75.644} C_DIS
LIN {X -0.079,Y -352.814,Z 1378.410,A 0.000,B 0.000,C 90.000,E1 73.866} C_DIS
LIN {X -0.204,Y -341.059,Z 1378.399,A 0.000,B 0.000,C 90.000,E1 71.764} C_DIS
LIN {X -0.041,Y -329.393,Z 1378.386,A 0.000,B 0.000,C 90.000,E1 69.571} C_DIS
LIN {X -0.080,Y -313.289,Z 1378.369,A 0.000,B 0.000,C 90.000,E1 66.410} C_DIS
LIN {X 0.041,Y -300.127,Z 1378.353,A 0.000,B 0.000,C 90.000,E1 63.461} C_DIS
LIN {X 0.071,Y -289.692,Z 1378.338,A 0.000,B 0.000,C 90.000,E1 60.795} C_DIS
LIN {X -0.107,Y -280.400,Z 1378.323,A 0.000,B 0.000,C 90.000,E1 58.122} C_DIS
LIN {X -0.159,Y -269.946,Z 1378.304,A 0.000,B 0.000,C 90.000,E1 54.689} C_DIS
LIN {X 0.126,Y -262.049,Z 1378.288,A 0.000,B 0.000,C 90.000,E1 51.823} C_DIS
LIN {X 0.001,Y -252.717,Z 1378.268,A 0.000,B 0.000,C 90.000,E1 48.286} C_DIS
LIN {X -0.079,Y -245.669,Z 1378.252,A 0.000,B 0.000,C 90.000,E1 45.405} C_DIS
LIN {X 0.123,Y -237.531,Z 1378.232,A 0.000,B 0.000,C 90.000,E1 41.676} C_DIS
LIN {X -0.020,Y -230.283,Z 1378.211,A 0.000,B 0.000,C 90.000,E1 37.971} C_DIS
LIN {X -0.111,Y -224.012,Z 1378.190,A 0.000,B 0.000,C 90.000,E1 34.199} C_DIS
LIN {X -0.032,Y -218.620,Z 1378.168,A 0.000,B 0.000,C 90.000,E1 30.335} C_DIS
LIN {X 0.013,Y -214.162,Z 1378.147,A 0.000,B 0.000,C 90.000,E1 26.437} C_DIS
LIN {X 0.055,Y -210.191,Z 1378.121,A 0.000,B 0.000,C 90.000,E1 21.716} C_DIS
LIN {X 0.001,Y -207.340,Z 1378.094,A 0.000,B 0.000,C 90.000,E1 16.985} C_DIS
LIN {X -0.082,Y -205.719,Z 1378.077,A 0.000,B 0.000,C 90.000,E1 13.828} C_DIS
LIN {X -0.055,Y -203.463,Z 1378.050,A 0.000,B 0.000,C 90.000,E1 9.029} C_DIS
LIN {X 0.042,Y -201.903,Z 1378.028,A 0.000,B 0.000,C 90.000,E1 4.992} C_DIS
LIN {X 0.025,Y -200.522,Z 1378.005,A 0.000,B 0.000,C 90.000,E1 0.974} C_DIS
LIN {X -0.089,Y -199.620,Z 1377.984,A 0.000,B 0.000,C 90.000,E1 357.135} C_DIS
LIN {X 0.064,Y -199.290,Z 1377.948,A 0.000,B 0.000,C 90.000,E1 350.622} C_DIS
LIN {X 0.069,Y -201.628,Z 1377.903,A 0.000,B 0.000,C 90.000,E1 342.543} C_DIS
LIN {X 0.082,Y -204.695,Z 1377.876,A 0.000,B 0.000,C 90.000,E1 337.720} C_DIS
LIN {X -0.056,Y -208.449,Z 1377.854,A 0.000,B 0.000,C 90.000,E1 333.768} C_DIS
LIN {X 0.014,Y -213.333,Z 1377.832,A 0.000,B 0.000,C 90.000,E1 329.793} C_DIS
LIN {X 0.013,Y -219.509,Z 1377.810,A 0.000,B 0.000,C 90.000,E1 325.881} C_DIS
LIN {X 0.113,Y -225.323,Z 1377.793,A 0.000,B 0.000,C 90.000,E1 322.763} C_DIS
LIN {X -0.037,Y -232.066,Z 1377.776,A 0.000,B 0.000,C 90.000,E1 319.747} C_DIS
LIN {X -0.099,Y -240.631,Z 1377.758,A 0.000,B 0.000,C 90.000,E1 316.377} C_DIS
LIN {X 0.091,Y -250.204,Z 1377.739,A 0.000,B 0.000,C 90.000,E1 313.014} C_DIS
LIN {X 0.017,Y -258.641,Z 1377.725,A 0.000,B 0.000,C 90.000,E1 310.496} C_DIS
LIN {X 0.021,Y -269.445,Z 1377.709,A 0.000,B 0.000,C 90.000,E1 307.649} C_DIS
LIN {X -0.095,Y -279.902,Z 1377.696,A 0.000,B 0.000,C 90.000,E1 305.231} C_DIS
LIN {X -0.005,Y -288.237,Z 1377.686,A 0.000,B 0.000,C 90.000,E1 303.499} C_DIS
LIN {X 0.060,Y -297.557,Z 1377.677,A 0.000,B 0.000,C 90.000,E1 301.799} C_DIS
LIN {X 0.099,Y -305.964,Z 1377.669,A 0.000,B 0.000,C 90.000,E1 300.463} C_DIS
LIN {X 0.094,Y -315.298,Z 1377.662,A 0.000,B 0.000,C 90.000,E1 299.155} C_DIS
LIN {X -0.059,Y -330.643,Z 1377.652,A 0.000,B 0.000,C 90.000,E1 297.308} C_DIS
LIN {X -0.076,Y -346.718,Z 1377.642,A 0.000,B 0.000,C 90.000,E1 295.515} C_DIS
LIN {X -0.184,Y -360.087,Z 1377.634,A 0.000,B 0.000,C 90.000,E1 294.079} C_DIS
LIN {X 0.120,Y -373.172,Z 1377.626,A 0.000,B 0.000,C 90.000,E1 292.589} C_DIS
LIN {X 0.031,Y -383.359,Z 1377.619,A 0.000,B 0.000,C 90.000,E1 291.461} C_DIS
LIN {X -0.109,Y -395.725,Z 1377.611,A 0.000,B 0.000,C 90.000,E1 290.047} C_DIS
LIN {X -0.144,Y -415.527,Z 1377.599,A 0.000,B 0.000,C 90.000,E1 287.819} C_DIS
LIN {X -0.054,Y -422.953,Z 1377.594,A 0.000,B 0.000,C 90.000,E1 286.985} C_DIS
LIN {X 0.104,Y -429.760,Z 1377.590,A 0.000,B 0.000,C 90.000,E1 286.150} C_DIS
LIN {X -0.096,Y -435.977,Z 1377.585,A 0.000,B 0.000,C 90.000,E1 285.371} C_DIS
LIN {X 0.183,Y -441.452,Z 1377.581,A 0.000,B 0.000,C 90.000,E1 284.537} C_DIS
LIN {X -0.030,Y -446.097,Z 1377.577,A 0.000,B 0.000,C 90.000,E1 283.772} C_DIS
LIN {X -0.198,Y -449.907,Z 1377.572,A 0.000,B 0.000,C 90.000,E1 283.008} C_DIS
LIN {X 0.105,Y -452.977,Z 1377.568,A 0.000,B 0.000,C 90.000,E1 282.187} C_DIS
LIN {X 0.172,Y -454.558,Z 1377.565,A 0.000,B 0.000,C 90.000,E1 281.658} C_DIS
LIN {X -0.197,Y -455.732,Z 1377.562,A 0.000,B 0.000,C 90.000,E1 281.186} C_DIS
LIN {X -0.113,Y -456.518,Z 1377.559,A 0.000,B 0.000,C 90.000,E1 280.658} C_DIS
LIN {X -0.104,Y -456.869,Z 1377.556,A 0.000,B 0.000,C 90.000,E1 280.141} C_DIS
LIN {X -0.010,Y -456.780,Z 1377.553,A 0.000,B 0.000,C 90.000,E1 279.613} C_DIS
LIN {X 0.010,Y -456.219,Z 1377.551,A 0.000,B 0.000,C 90.000,E1 279.095} C_DIS
LIN {X 0.101,Y -455.194,Z 1377.548,A 0.000,B 0.000,C 90.000,E1 278.568} C_DIS
LIN {X 0.119,Y -453.665,Z 1377.545,A 0.000,B 0.000,C 90.000,E1 278.049} C_DIS
LIN {X 0.133,Y -451.613,Z 1377.542,A 0.000,B 0.000,C 90.000,E1 277.530} C_DIS
LIN {X 0.140,Y -448.976,Z 1377.539,A 0.000,B 0.000,C 90.000,E1 277.011} C_DIS
LIN {X 0.179,Y -445.677,Z 1377.536,A 0.000,B 0.000,C 90.000,E1 276.486} C_DIS
LIN {X 0.146,Y -441.500,Z 1377.533,A 0.000,B 0.000,C 90.000,E1 275.967} C_DIS
LIN {X 0.051,Y -436.262,Z 1377.530,A 0.000,B 0.000,C 90.000,E1 275.454} C_DIS
LIN {X -0.180,Y -430.264,Z 1377.528,A 0.000,B 0.000,C 90.000,E1 274.992} C_DIS
LIN {X 0.041,Y -423.931,Z 1377.525,A 0.000,B 0.000,C 90.000,E1 274.531} C_DIS
LIN {X 0.178,Y -417.327,Z 1377.523,A 0.000,B 0.000,C 90.000,E1 274.131} C_DIS
LIN {X -0.121,Y -410.594,Z 1377.521,A 0.000,B 0.000,C 90.000,E1 273.841} C_DIS
LIN {X 0.133,Y -400.722,Z 1377.519,A 0.000,B 0.000,C 90.000,E1 273.383} C_DIS
LIN {X -0.044,Y -390.694,Z 1377.517,A 0.000,B 0.000,C 90.000,E1 273.037} C_DIS
LIN {X 0.132,Y -380.514,Z 1377.515,A 0.000,B 0.000,C 90.000,E1 272.694} C_DIS
LIN {X -0.087,Y -369.642,Z 1377.514,A 0.000,B 0.000,C 90.000,E1 272.465} C_DIS
LIN {X 0.108,Y -357.976,Z 1377.513,A 0.000,B 0.000,C 90.000,E1 272.236} C_DIS
LIN {X 0.153,Y -349.305,Z 1377.512,A 0.000,B 0.000,C 90.000,E1 272.121} C_DIS
LIN {X -0.146,Y -333.998,Z 1377.511,A 0.000,B 0.000,C 90.000,E1 272.064} C_DIS
LIN {X 0.030,Y -322.632,Z 1377.511,A 0.000,B 0.000,C 90.000,E1 272.007} C_DIS
LIN {X -0.008,Y -181.261,Z 1377.511,A 0.000,B 0.000,C 90.000,E1 272.007} C_DIS
LIN {X -0.036,Y -181.581,Z 1377.502,A 0.000,B 0.000,C 90.000,E1 270.286} C_DIS
LIN {X -0.061,Y -180.898,Z 1377.474,A 0.000,B 0.000,C 90.000,E1 265.241} C_DIS
LIN {X -0.038,Y -179.849,Z 1377.459,A 0.000,B 0.000,C 90.000,E1 262.704} C_DIS
LIN {X 0.019,Y -179.030,Z 1377.445,A 0.000,B 0.000,C 90.000,E1 260.151} C_DIS
LIN {X -0.095,Y -178.682,Z 1377.441,A 0.000,B 0.000,C 90.000,E1 259.342} C_DIS
LIN {X 0.016,Y -175.732,Z 1377.412,A 0.000,B 0.000,C 90.000,E1 254.212} C_DIS
LIN {X 0.012,Y -171.917,Z 1377.384,A 0.000,B 0.000,C 90.000,E1 249.082} C_DIS
LIN {X -0.013,Y -171.285,Z 1377.379,A 0.000,B 0.000,C 90.000,E1 248.230} C_DIS
LIN {X 0.034,Y -167.551,Z 1377.355,A 0.000,B 0.000,C 90.000,E1 243.896} C_DIS
LIN {X 0.047,Y -166.171,Z 1377.345,A 0.000,B 0.000,C 90.000,E1 242.153} C_DIS
LIN {X 0.036,Y -162.944,Z 1377.326,A 0.000,B 0.000,C 90.000,E1 238.663} C_DIS
LIN {X 0.014,Y -161.614,Z 1377.316,A 0.000,B 0.000,C 90.000,E1 236.914} C_DIS
LIN {X -0.011,Y -159.142,Z 1377.302,A 0.000,B 0.000,C 90.000,E1 234.276} C_DIS
LIN {X 0.000,Y -155.663,Z 1377.277,A 0.000,B 0.000,C 90.000,E1 229.828} C_DIS
LIN {X 0.052,Y -151.932,Z 1377.252,A 0.000,B 0.000,C 90.000,E1 225.324} C_DIS
LIN {X 0.066,Y -150.169,Z 1377.237,A 0.000,B 0.000,C 90.000,E1 222.609} C_DIS
LIN {X -0.013,Y -146.947,Z 1377.212,A 0.000,B 0.000,C 90.000,E1 218.096} C_DIS
LIN {X -0.026,Y -145.534,Z 1377.196,A 0.000,B 0.000,C 90.000,E1 215.358} C_DIS
LIN {X 0.014,Y -142.931,Z 1377.171,A 0.000,B 0.000,C 90.000,E1 210.747} C_DIS
LIN {X 0.013,Y -141.555,Z 1377.150,A 0.000,B 0.000,C 90.000,E1 207.052} C_DIS
LIN {X 0.002,Y -139.407,Z 1377.114,A 0.000,B 0.000,C 90.000,E1 200.556} C_DIS
LIN {X -0.076,Y -139.126,Z 1377.104,A 0.000,B 0.000,C 90.000,E1 198.725} C_DIS
LIN {X -0.049,Y -138.351,Z 1377.057,A 0.000,B 0.000,C 90.000,E1 190.310} C_DIS
LIN {X -0.062,Y -139.500,Z 1377.005,A 0.000,B 0.000,C 90.000,E1 180.974} C_DIS
LIN {X 0.019,Y -141.125,Z 1376.974,A 0.000,B 0.000,C 90.000,E1 175.355} C_DIS
LIN {X -0.029,Y -142.505,Z 1376.959,A 0.000,B 0.000,C 90.000,E1 172.591} C_DIS
LIN {X 0.060,Y -144.762,Z 1376.933,A 0.000,B 0.000,C 90.000,E1 167.937} C_DIS
LIN {X 0.009,Y -147.373,Z 1376.913,A 0.000,B 0.000,C 90.000,E1 164.283} C_DIS
LIN {X 0.072,Y -150.701,Z 1376.887,A 0.000,B 0.000,C 90.000,E1 159.699} C_DIS
LIN {X 0.013,Y -154.182,Z 1376.867,A 0.000,B 0.000,C 90.000,E1 156.102} C_DIS
LIN {X -0.057,Y -157.617,Z 1376.847,A 0.000,B 0.000,C 90.000,E1 152.538} C_DIS
LIN {X 0.031,Y -161.873,Z 1376.828,A 0.000,B 0.000,C 90.000,E1 148.948} C_DIS
LIN {X 0.004,Y -166.063,Z 1376.808,A 0.000,B 0.000,C 90.000,E1 145.435} C_DIS
LIN {X 0.005,Y -171.068,Z 1376.789,A 0.000,B 0.000,C 90.000,E1 141.949} C_DIS
LIN {X 0.061,Y -175.941,Z 1376.770,A 0.000,B 0.000,C 90.000,E1 138.485} C_DIS
LIN {X -0.079,Y -180.182,Z 1376.755,A 0.000,B 0.000,C 90.000,E1 135.972} C_DIS
LIN {X -0.111,Y -185.599,Z 1376.737,A 0.000,B 0.000,C 90.000,E1 132.609} C_DIS
LIN {X -0.062,Y -190.191,Z 1376.723,A 0.000,B 0.000,C 90.000,E1 130.092} C_DIS
LIN {X -0.018,Y -197.520,Z 1376.700,A 0.000,B 0.000,C 90.000,E1 125.964} C_DIS
LIN {X -0.088,Y -199.276,Z 1376.695,A 0.000,B 0.000,C 90.000,E1 125.105} C_DIS
LIN {X -0.172,Y -309.001,Z 1376.695,A 0.000,B 0.000,C 90.000,E1 125.105} C_DIS
LIN {X -0.052,Y -312.198,Z 1376.695,A 0.000,B 0.000,C 90.000,E1 125.025} C_DIS
LIN {X -0.098,Y -317.813,Z 1376.693,A 0.000,B 0.000,C 90.000,E1 124.692} C_DIS
LIN {X 0.038,Y -320.842,Z 1376.691,A 0.000,B 0.000,C 90.000,E1 124.326} C_DIS
LIN {X -0.070,Y -322.802,Z 1376.689,A 0.000,B 0.000,C 90.000,E1 124.040} C_DIS
LIN {X 0.089,Y -324.328,Z 1376.687,A 0.000,B 0.000,C 90.000,E1 123.706} C_DIS
LIN {X 0.100,Y -327.773,Z 1376.682,A 0.000,B 0.000,C 90.000,E1 122.752} C_DIS
LIN {X -0.018,Y -338.444,Z 1376.666,A 0.000,B 0.000,C 90.000,E1 119.951} C_DIS
LIN {X -0.005,Y -350.471,Z 1376.651,A 0.000,B 0.000,C 90.000,E1 117.180} C_DIS
LIN {X 0.018,Y -363.965,Z 1376.636,A 0.000,B 0.000,C 90.000,E1 114.463} C_DIS
LIN {X 0.038,Y -377.280,Z 1376.623,A 0.000,B 0.000,C 90.000,E1 112.099} C_DIS
LIN {X -0.112,Y -391.936,Z 1376.610,A 0.000,B 0.000,C 90.000,E1 109.812} C_DIS
LIN {X 0.197,Y -408.036,Z 1376.597,A 0.000,B 0.000,C 90.000,E1 107.511} C_DIS
LIN {X -0.242,Y -425.691,Z 1376.585,A 0.000,B 0.000,C 90.000,E1 105.371} C_DIS
LIN {X 0.205,Y -444.972,Z 1376.573,A 0.000,B 0.000,C 90.000,E1 103.175} C_DIS
LIN {X 0.214,Y -465.111,Z 1376.562,A 0.000,B 0.000,C 90.000,E1 101.186} C_DIS
LIN {X -0.053,Y -483.012,Z 1376.553,A 0.000,B 0.000,C 90.000,E1 99.613} C_DIS
LIN {X 0.066,Y -484.884,Z 1376.552,A 0.000,B 0.000,C 90.000,E1 99.378} C_DIS
LIN {X -0.125,Y -486.479,Z 1376.551,A 0.000,B 0.000,C 90.000,E1 99.151} C_DIS
LIN {X -0.239,Y -487.673,Z 1376.549,A 0.000,B 0.000,C 90.000,E1 98.916} C_DIS
LIN {X -0.040,Y -489.113,Z 1376.547,A 0.000,B 0.000,C 90.000,E1 98.398} C_DIS
LIN {X 0.237,Y -489.505,Z 1376.544,A 0.000,B 0.000,C 90.000,E1 97.871} C_DIS
LIN {X -0.033,Y -488.913,Z 1376.541,A 0.000,B 0.000,C 90.000,E1 97.409} C_DIS
LIN {X 0.184,Y -487.241,Z 1376.538,A 0.000,B 0.000,C 90.000,E1 96.891} C_DIS
LIN {X 0.022,Y -485.907,Z 1376.537,A 0.000,B 0.000,C 90.000,E1 96.663} C_DIS
LIN {X -0.080,Y -473.917,Z 1376.527,A 0.000,B 0.000,C 90.000,E1 94.935} C_DIS
LIN {X 0.016,Y -462.567,Z 1376.518,A 0.000,B 0.000,C 90.000,E1 93.154} C_DIS
LIN {X 0.056,Y -445.959,Z 1376.503,A 0.000,B 0.000,C 90.000,E1 90.573} C_DIS
LIN {X 0.058,Y -430.860,Z 1376.489,A 0.000,B 0.000,C 90.000,E1 87.936} C_DIS
LIN {X -0.139,Y -418.982,Z 1376.477,A 0.000,B 0.000,C 90.000,E1 85.812} C_DIS
LIN {X 0.176,Y -408.405,Z 1376.466,A 0.000,B 0.000,C 90.000,E1 83.856} C_DIS
LIN {X -0.181,Y -399.206,Z 1376.457,A 0.000,B 0.000,C 90.000,E1 82.243} C_DIS
LIN {X 0.196,Y -389.857,Z 1376.447,A 0.000,B 0.000,C 90.000,E1 80.500} C_DIS
LIN {X 0.019,Y -380.327,Z 1376.438,A 0.000,B 0.000,C 90.000,E1 78.814} C_DIS
LIN {X 0.105,Y -369.031,Z 1376.427,A 0.000,B 0.000,C 90.000,E1 76.769} C_DIS
LIN {X 0.154,Y -359.189,Z 1376.417,A 0.000,B 0.000,C 90.000,E1 74.991} C_DIS
LIN {X 0.127,Y -349.168,Z 1376.407,A 0.000,B 0.000,C 90.000,E1 73.196} C_DIS
LIN {X -0.073,Y -337.434,Z 1376.395,A 0.000,B 0.000,C 90.000,E1 71.094} C_DIS
LIN {X -0.024,Y -324.193,Z 1376.381,A 0.000,B 0.000,C 90.000,E1 68.592} C_DIS
LIN {X -0.145,Y -309.991,Z 1376.365,A 0.000,B 0.000,C 90.000,E1 65.741} C_DIS
LIN {X -0.140,Y -298.533,Z 1376.351,A 0.000,B 0.000,C 90.000,E1 63.127} C_DIS
LIN {X -0.137,Y -288.282,Z 1376.336,A 0.000,B 0.000,C 90.000,E1 60.461} C_DIS
LIN {X -0.064,Y -280.230,Z 1376.323,A 0.000,B 0.000,C 90.000,E1 58.074} C_DIS
LIN {X 0.025,Y -269.830,Z 1376.303,A 0.000,B 0.000,C 90.000,E1 54.609} C_DIS
LIN {X -0.064,Y -261.978,Z 1376.288,A 0.000,B 0.000,C 90.000,E1 51.823} C_DIS
LIN {X 0.005,Y -252.674,Z 1376.268,A 0.000,B 0.000,C 90.000,E1 48.243} C_DIS
LIN {X 0.087,Y -245.644,Z 1376.252,A 0.000,B 0.000,C 90.000,E1 45.324} C_DIS
LIN {X -0.052,Y -237.545,Z 1376.231,A 0.000,B 0.000,C 90.000,E1 41.676} C_DIS
LIN {X -0.049,Y -230.326,Z 1376.211,A 0.000,B 0.000,C 90.000,E1 37.935} C_DIS
LIN {X 0.037,Y -224.075,Z 1376.190,A 0.000,B 0.000,C 90.000,E1 34.119} C_DIS
LIN {X 0.111,Y -218.719,Z 1376.168,A 0.000,B 0.000,C 90.000,E1 30.256} C_DIS
LIN {X -0.042,Y -214.307,Z 1376.147,A 0.000,B 0.000,C 90.000,E1 26.411} C_DIS
LIN {X -0.087,Y -210.371,Z 1376.120,A 0.000,B 0.000,C 90.000,E1 21.716} C_DIS
LIN {X -0.084,Y -207.974,Z 1376.099,A 0.000,B 0.000,C 90.000,E1 17.764} C_DIS
LIN {X 0.104,Y -206.306,Z 1376.081,A 0.000,B 0.000,C 90.000,E1 14.537} C_DIS
LIN {X 0.043,Y -204.685,Z 1376.063,A 0.000,B 0.000,C 90.000,E1 11.366} C_DIS
LIN {X 0.094,Y -202.973,Z 1376.041,A 0.000,B 0.000,C 90.000,E1 7.352} C_DIS
LIN {X -0.066,Y -201.747,Z 1376.023,A 0.000,B 0.000,C 90.000,E1 4.188} C_DIS
LIN {X -0.037,Y -200.282,Z 1375.997,A 0.000,B 0.000,C 90.000,E1 359.542} C_DIS
LIN {X 0.073,Y -199.403,Z 1375.970,A 0.000,B 0.000,C 90.000,E1 354.666} C_DIS
LIN {X -0.039,Y -199.787,Z 1375.935,A 0.000,B 0.000,C 90.000,E1 348.229} C_DIS
LIN {X -0.002,Y -202.217,Z 1375.899,A 0.000,B 0.000,C 90.000,E1 341.764} C_DIS
LIN {X 0.102,Y -205.536,Z 1375.872,A 0.000,B 0.000,C 90.000,E1 336.922} C_DIS
LIN {X -0.115,Y -209.534,Z 1375.850,A 0.000,B 0.000,C 90.000,E1 332.999} C_DIS
LIN {X 0.092,Y -214.666,Z 1375.828,A 0.000,B 0.000,C 90.000,E1 328.997} C_DIS
LIN {X 0.073,Y -221.095,Z 1375.806,A 0.000,B 0.000,C 90.000,E1 325.102} C_DIS
LIN {X 0.037,Y -227.091,Z 1375.789,A 0.000,B 0.000,C 90.000,E1 322.029} C_DIS
LIN {X -0.071,Y -234.057,Z 1375.772,A 0.000,B 0.000,C 90.000,E1 319.013} C_DIS
LIN {X -0.091,Y -242.809,Z 1375.754,A 0.000,B 0.000,C 90.000,E1 315.648} C_DIS
LIN {X -0.002,Y -252.637,Z 1375.735,A 0.000,B 0.000,C 90.000,E1 312.324} C_DIS
LIN {X 0.019,Y -262.662,Z 1375.719,A 0.000,B 0.000,C 90.000,E1 309.439} C_DIS
LIN {X 0.173,Y -273.925,Z 1375.703,A 0.000,B 0.000,C 90.000,E1 306.583} C_DIS
LIN {X 0.050,Y -283.238,Z 1375.692,A 0.000,B 0.000,C 90.000,E1 304.532} C_DIS
LIN {X 0.040,Y -291.953,Z 1375.682,A 0.000,B 0.000,C 90.000,E1 302.832} C_DIS
LIN {X 0.166,Y -299.624,Z 1375.675,A 0.000,B 0.000,C 90.000,E1 301.465} C_DIS
LIN {X -0.030,Y -308.278,Z 1375.668,A 0.000,B 0.000,C 90.000,E1 300.178} C_DIS
LIN {X 0.021,Y -317.808,Z 1375.660,A 0.000,B 0.000,C 90.000,E1 298.871} C_DIS
LIN {X 0.119,Y -341.262,Z 1375.645,A 0.000,B 0.000,C 90.000,E1 296.104} C_DIS
LIN {X -0.064,Y -357.216,Z 1375.635,A 0.000,B 0.000,C 90.000,E1 294.387} C_DIS
LIN {X -0.134,Y -370.389,Z 1375.627,A 0.000,B 0.000,C 90.000,E1 292.950} C_DIS
LIN {X 0.048,Y -380.719,Z 1375.621,A 0.000,B 0.000,C 90.000,E1 291.770} C_DIS
LIN {X -0.110,Y -393.177,Z 1375.613,A 0.000,B 0.000,C 90.000,E1 290.355} C_DIS
LIN {X -0.111,Y -412.929,Z 1375.600,A 0.000,B 0.000,C 90.000,E1 288.109} C_DIS
LIN {X 0.156,Y -422.775,Z 1375.594,A 0.000,B 0.000,C 90.000,E1 286.985} C_DIS
LIN {X 0.183,Y -431.760,Z 1375.589,A 0.000,B 0.000,C 90.000,E1 285.898} C_DIS
LIN {X -0.114,Y -437.794,Z 1375.584,A 0.000,B 0.000,C 90.000,E1 285.134} C_DIS
LIN {X -0.029,Y -441.391,Z 1375.581,A 0.000,B 0.000,C 90.000,E1 284.592} C_DIS
LIN {X 0.186,Y -446.092,Z 1375.577,A 0.000,B 0.000,C 90.000,E1 283.772} C_DIS
LIN {X 0.020,Y -449.962,Z 1375.572,A 0.000,B 0.000,C 90.000,E1 283.008} C_DIS
LIN {X -0.118,Y -453.085,Z 1375.568,A 0.000,B 0.000,C 90.000,E1 282.243} C_DIS
LIN {X -0.052,Y -454.713,Z 1375.565,A 0.000,B 0.000,C 90.000,E1 281.715} C_DIS
LIN {X 0.025,Y -455.929,Z 1375.562,A 0.000,B 0.000,C 90.000,E1 281.186} C_DIS
LIN {X 0.110,Y -456.731,Z 1375.559,A 0.000,B 0.000,C 90.000,E1 280.658} C_DIS
LIN {X 0.120,Y -457.105,Z 1375.556,A 0.000,B 0.000,C 90.000,E1 280.141} C_DIS
LIN {X 0.215,Y -457.072,Z 1375.554,A 0.000,B 0.000,C 90.000,E1 279.613} C_DIS
LIN {X -0.214,Y -456.566,Z 1375.551,A 0.000,B 0.000,C 90.000,E1 279.151} C_DIS
LIN {X -0.121,Y -455.535,Z 1375.548,A 0.000,B 0.000,C 90.000,E1 278.624} C_DIS
LIN {X -0.101,Y -454.068,Z 1375.545,A 0.000,B 0.000,C 90.000,E1 278.106} C_DIS
LIN {X -0.084,Y -452.034,Z 1375.542,A 0.000,B 0.000,C 90.000,E1 277.587} C_DIS
LIN {X -0.075,Y -449.479,Z 1375.539,A 0.000,B 0.000,C 90.000,E1 277.068} C_DIS
LIN {X -0.082,Y -446.241,Z 1375.536,A 0.000,B 0.000,C 90.000,E1 276.549} C_DIS
LIN {X -0.106,Y -442.230,Z 1375.533,A 0.000,B 0.000,C 90.000,E1 276.030} C_DIS
LIN {X -0.150,Y -437.171,Z 1375.531,A 0.000,B 0.000,C 90.000,E1 275.511} C_DIS
LIN {X -0.048,Y -431.145,Z 1375.528,A 0.000,B 0.000,C 90.000,E1 274.992} C_DIS
LIN {X 0.123,Y -424.818,Z 1375.525,A 0.000,B 0.000,C 90.000,E1 274.531} C_DIS
LIN {X -0.104,Y -418.541,Z 1375.523,A 0.000,B 0.000,C 90.000,E1 274.188} C_DIS
LIN {X 0.115,Y -408.516,Z 1375.521,A 0.000,B 0.000,C 90.000,E1 273.669} C_DIS
LIN {X 0.009,Y -398.524,Z 1375.518,A 0.000,B 0.000,C 90.000,E1 273.269} C_DIS
LIN {X -0.061,Y -388.480,Z 1375.516,A 0.000,B 0.000,C 90.000,E1 272.922} C_DIS
LIN {X 0.062,Y -381.521,Z 1375.515,A 0.000,B 0.000,C 90.000,E1 272.694} C_DIS
LIN {X -0.008,Y -374.308,Z 1375.514,A 0.000,B 0.000,C 90.000,E1 272.522} C_DIS
LIN {X 0.052,Y -362.791,Z 1375.513,A 0.000,B 0.000,C 90.000,E1 272.293} C_DIS
LIN {X 0.085,Y -350.361,Z 1375.512,A 0.000,B 0.000,C 90.000,E1 272.121} C_DIS
LIN {X 0.113,Y -334.738,Z 1375.511,A 0.000,B 0.000,C 90.000,E1 272.007} C_DIS
LIN {X -0.047,Y -324.023,Z 1375.511,A 0.000,B 0.000,C 90.000,E1 272.007} C_DIS
LIN {X -0.051,Y -181.263,Z 1375.511,A 0.000,B 0.000,C 90.000,E1 272.007} C_DIS
LIN {X -0.082,Y -181.581,Z 1375.501,A 0.000,B 0.000,C 90.000,E1 270.286} C_DIS
LIN {X 0.073,Y -180.896,Z 1375.473,A 0.000,B 0.000,C 90.000,E1 265.184} C_DIS
LIN {X -0.083,Y -179.842,Z 1375.459,A 0.000,B 0.000,C 90.000,E1 262.704} C_DIS
LIN {X -0.027,Y -179.027,Z 1375.445,A 0.000,B 0.000,C 90.000,E1 260.151} C_DIS
LIN {X 0.035,Y -178.674,Z 1375.441,A 0.000,B 0.000,C 90.000,E1 259.285} C_DIS
LIN {X -0.029,Y -175.723,Z 1375.412,A 0.000,B 0.000,C 90.000,E1 254.212} C_DIS
LIN {X -0.012,Y -172.440,Z 1375.389,A 0.000,B 0.000,C 90.000,E1 249.934} C_DIS
LIN {X -0.057,Y -171.271,Z 1375.379,A 0.000,B 0.000,C 90.000,E1 248.230} C_DIS
LIN {X -0.011,Y -167.540,Z 1375.355,A 0.000,B 0.000,C 90.000,E1 243.896} C_DIS
LIN {X 0.003,Y -166.156,Z 1375.345,A 0.000,B 0.000,C 90.000,E1 242.153} C_DIS
LIN {X -0.006,Y -162.932,Z 1375.326,A 0.000,B 0.000,C 90.000,E1 238.663} C_DIS
LIN {X -0.029,Y -161.604,Z 1375.316,A 0.000,B 0.000,C 90.000,E1 236.914} C_DIS
LIN {X -0.052,Y -159.129,Z 1375.301,A 0.000,B 0.000,C 90.000,E1 234.276} C_DIS
LIN {X -0.043,Y -155.650,Z 1375.277,A 0.000,B 0.000,C 90.000,E1 229.828} C_DIS
LIN {X 0.010,Y -151.922,Z 1375.252,A 0.000,B 0.000,C 90.000,E1 225.324} C_DIS
LIN {X 0.026,Y -150.156,Z 1375.237,A 0.000,B 0.000,C 90.000,E1 222.609} C_DIS
LIN {X -0.053,Y -146.937,Z 1375.212,A 0.000,B 0.000,C 90.000,E1 218.096} C_DIS
LIN {X 0.054,Y -145.525,Z 1375.196,A 0.000,B 0.000,C 90.000,E1 215.311} C_DIS
LIN {X 0.048,Y -142.924,Z 1375.171,A 0.000,B 0.000,C 90.000,E1 210.718} C_DIS
LIN {X -0.026,Y -141.547,Z 1375.150,A 0.000,B 0.000,C 90.000,E1 207.052} C_DIS
LIN {X -0.037,Y -139.404,Z 1375.114,A 0.000,B 0.000,C 90.000,E1 200.556} C_DIS
LIN {X 0.016,Y -139.122,Z 1375.104,A 0.000,B 0.000,C 90.000,E1 198.671} C_DIS
LIN {X 0.049,Y -138.351,Z 1375.057,A 0.000,B 0.000,C 90.000,E1 190.254} C_DIS
LIN {X 0.038,Y -139.502,Z 1375.005,A 0.000,B 0.000,C 90.000,E1 180.917} C_DIS
LIN {X -0.021,Y -141.132,Z 1374.974,A 0.000,B 0.000,C 90.000,E1 175.355} C_DIS
LIN {X -0.068,Y -142.512,Z 1374.959,A 0.000,B 0.000,C 90.000,E1 172.591} C_DIS
LIN {X 0.019,Y -144.772,Z 1374.933,A 0.000,B 0.000,C 90.000,E1 167.937} C_DIS
LIN {X -0.031,Y -147.385,Z 1374.913,A 0.000,B 0.000,C 90.000,E1 164.283} C_DIS
LIN {X 0.030,Y -150.715,Z 1374.887,A 0.000,B 0.000,C 90.000,E1 159.699} C_DIS
LIN {X -0.029,Y -154.196,Z 1374.867,A 0.000,B 0.000,C 90.000,E1 156.102} C_DIS
LIN {X 0.041,Y -157.634,Z 1374.847,A 0.000,B 0.000,C 90.000,E1 152.487} C_DIS
LIN {X -0.012,Y -161.892,Z 1374.828,A 0.000,B 0.000,C 90.000,E1 148.948} C_DIS
LIN {X 0.097,Y -166.082,Z 1374.808,A 0.000,B 0.000,C 90.000,E1 145.388} C_DIS
LIN {X 0.096,Y -171.090,Z 1374.789,A 0.000,B 0.000,C 90.000,E1 141.904} C_DIS
LIN {X 0.016,Y -175.964,Z 1374.769,A 0.000,B 0.000,C 90.000,E1 138.485} C_DIS
LIN {X 0.005,Y -180.208,Z 1374.755,A 0.000,B 0.000,C 90.000,E1 135.931} C_DIS
